// Check ParCmd.Offset.Config.Shoulder valid ? 
IF (( ParCmd.Offset.Config.Shoulder <> ArmConfigShoulder.USE_CONFIG ) AND  
    ( ParCmd.Offset.Config.Shoulder <> ArmConfigShoulder.SAME       ) AND
    ( ParCmd.Offset.Config.Shoulder <> ArmConfigShoulder.FREE       ) AND
    ( ParCmd.Offset.Config.Shoulder <> ArmConfigShoulder.BACK       ) AND
    ( ParCmd.Offset.Config.Shoulder <> ArmConfigShoulder.FRONT      ))
THEN
  // Parameter not valid
  CheckParameterValid := FALSE;
  // Set error
  SetError( ErrorID := RobotLibraryErrorIdEnum.ERR_CONFIGMODE_SHOULDER_INVALID, Overwrite := TRUE );
  // Create log entry
  CreateLogMessagePara1 ( Timestamp   := AxesGroup.State.SystemTime,
                          MessageType := MessageType.CMD,
                          Severity    := Severity.ERROR,
                          MessageCode := ErrorID,
                          MessageText := 'Invalid Parameter ParCmd.Offset.Config.Shoulder = {1}',
                          Para1       :=  ARM_CONFIG_SHOULDER_TO_STRING(ParCmd.Offset.Config.Shoulder));
  RETURN;                          
END_IF


// Check ParCmd.Offset.Config.Elbow valid ? 
IF (( ParCmd.Offset.Config.Elbow <> ArmConfigElbow.USE_CONFIG ) AND  
    ( ParCmd.Offset.Config.Elbow <> ArmConfigElbow.SAME       ) AND
    ( ParCmd.Offset.Config.Elbow <> ArmConfigElbow.FREE       ) AND
    ( ParCmd.Offset.Config.Elbow <> ArmConfigElbow.DOWN       ) AND
    ( ParCmd.Offset.Config.Elbow <> ArmConfigElbow.UP         ))
THEN
  // Parameter not valid
  CheckParameterValid := FALSE;
  // Set error
  SetError( ErrorID := RobotLibraryErrorIdEnum.ERR_CONFIGMODE_ELBOW_INVALID, Overwrite := TRUE );
  // Create log entry
  CreateLogMessagePara1 ( Timestamp   := AxesGroup.State.SystemTime,
                          MessageType := MessageType.CMD,
                          Severity    := Severity.ERROR,
                          MessageCode := ErrorID,
                          MessageText := 'Invalid Parameter ParCmd.Offset.Config.Elbow = {1}',
                          Para1       :=  ARM_CONFIG_ELBOW_TO_STRING(ParCmd.Offset.Config.Elbow));
  RETURN;                          
END_IF


// Check ParCmd.Offset.Config.Wrist valid ? 
IF (( ParCmd.Offset.Config.Wrist <> ArmConfigWrist.USE_CONFIG ) AND  
    ( ParCmd.Offset.Config.Wrist <> ArmConfigWrist.SAME       ) AND
    ( ParCmd.Offset.Config.Wrist <> ArmConfigWrist.FREE       ) AND
    ( ParCmd.Offset.Config.Wrist <> ArmConfigWrist.FLIP       ) AND
    ( ParCmd.Offset.Config.Wrist <> ArmConfigWrist.NON_FLIP   ))
THEN
  // Parameter not valid
  CheckParameterValid := FALSE;
  // Set error
  SetError( ErrorID := RobotLibraryErrorIdEnum.ERR_CONFIGMODE_WRIST_INVALID, Overwrite := TRUE );
  // Create log entry
  CreateLogMessagePara1 ( Timestamp   := AxesGroup.State.SystemTime,
                          MessageType := MessageType.CMD,
                          Severity    := Severity.ERROR,
                          MessageCode := ErrorID,
                          MessageText := 'Invalid Parameter ParCmd.Offset.Config.Wrist = {1}',
                          Para1       :=  ARM_CONFIG_WRIST_TO_STRING(ParCmd.Offset.Config.Wrist));
  RETURN;                          
END_IF


// Check ParCmd.ReferenceType valid ? 
IF (( ParCmd.ReferenceType <> ReferenceType.TOOL  ) AND
    ( ParCmd.ReferenceType <> ReferenceType.FRAME ))  
THEN
  // Parameter not valid
  CheckParameterValid := FALSE;
  // Set error
  SetError( ErrorID := RobotLibraryErrorIdEnum.ERR_INVALID_PAR_CMD, Overwrite := TRUE );
  // Create log entry
  CreateLogMessagePara1 ( Timestamp   := AxesGroup.State.SystemTime,
                          MessageType := MessageType.CMD,
                          Severity    := Severity.ERROR,
                          MessageCode := ErrorID,
                          MessageText := 'Invalid Parameter ParCmd.ReferenceType = {1}',
                          Para1       := REFERENCE_TYPE_TO_STRING(ParCmd.ReferenceType));
  RETURN;                          
END_IF


// Check ParCmd.VelocityDiffRate valid ? 
IF  (( SysDepIsValidReal(ParCmd.VelocityDiffRate) = FALSE )  OR
    ((                   ParCmd.VelocityDiffRate  <     0 )  AND 
     (                   ParCmd.VelocityDiffRate <>    -1 )) OR   
     (                   ParCmd.VelocityDiffRate  >   100 ))      
THEN
  // Parameter not valid
  CheckParameterValid := FALSE;
  // Set error
  SetError( ErrorID := RobotLibraryErrorIdEnum.ERR_INVALID_PAR_CMD, Overwrite := TRUE );
  // Create log entry
  CreateLogMessagePara1 ( Timestamp   := AxesGroup.State.SystemTime,
                          MessageType := MessageType.CMD,
                          Severity    := Severity.ERROR,
                          MessageCode := ErrorID,
                          MessageText := 'Invalid Parameter ParCmd.VelocityDiffRate = {1}',
                          Para1       := VALID_REAL_TO_STRING(ParCmd.VelocityDiffRate));                            
  RETURN;
END_IF


// Check ParCmd.AccelerationDiffRate valid ? 
IF  (( SysDepIsValidReal(ParCmd.AccelerationDiffRate) = FALSE )  OR
    ((                   ParCmd.AccelerationDiffRate  <     0 )  AND 
     (                   ParCmd.AccelerationDiffRate <>    -1 )) OR   
     (                   ParCmd.AccelerationDiffRate  >   100 ))      
THEN
  // Parameter not valid
  CheckParameterValid := FALSE;
  // Set error
  SetError( ErrorID := RobotLibraryErrorIdEnum.ERR_ACCELERATION_INVALID, Overwrite := TRUE );
  // Create log entry
  CreateLogMessagePara1 ( Timestamp   := AxesGroup.State.SystemTime,
                          MessageType := MessageType.CMD,
                          Severity    := Severity.ERROR,
                          MessageCode := ErrorID,
                          MessageText := 'Invalid Parameter ParCmd.AccelerationDiffRate = {1}',
                          Para1       := VALID_REAL_TO_STRING(ParCmd.AccelerationDiffRate));                            
  RETURN;
END_IF


// Check ParCmd.DecelerationDiffRate valid ? 
IF  (( SysDepIsValidReal(ParCmd.DecelerationDiffRate) = FALSE )  OR
    ((                   ParCmd.DecelerationDiffRate  <     0 )  AND 
     (                   ParCmd.DecelerationDiffRate <>    -1 )) OR   
     (                   ParCmd.DecelerationDiffRate  >   100 ))      
THEN
  // Parameter not valid
  CheckParameterValid := FALSE;
  // Set error
  SetError( ErrorID := RobotLibraryErrorIdEnum.ERR_DECELERATION_INVALID, Overwrite := TRUE );
  // Create log entry
  CreateLogMessagePara1 ( Timestamp   := AxesGroup.State.SystemTime,
                          MessageType := MessageType.CMD,
                          Severity    := Severity.ERROR,
                          MessageCode := ErrorID,
                          MessageText := 'Invalid Parameter ParCmd.DecelerationDiffRate = {1}',
                          Para1       := VALID_REAL_TO_STRING(ParCmd.DecelerationDiffRate));                            
  RETURN;
END_IF


// Check ParCmd.JerkDiffRate valid ? 
IF  (( SysDepIsValidReal(ParCmd.JerkDiffRate) = FALSE )  OR
    ((                   ParCmd.JerkDiffRate  <     0 )  AND 
     (                   ParCmd.JerkDiffRate <>    -1 )) OR   
     (                   ParCmd.JerkDiffRate  >   100 ))      
THEN
  // Parameter not valid
  CheckParameterValid := FALSE;
  // Set error
  SetError( ErrorID := RobotLibraryErrorIdEnum.ERR_JERK_INVALID, Overwrite := TRUE );
  // Create log entry
  CreateLogMessagePara1 ( Timestamp   := AxesGroup.State.SystemTime,
                          MessageType := MessageType.CMD,
                          Severity    := Severity.ERROR,
                          MessageCode := ErrorID,
                          MessageText := 'Invalid Parameter ParCmd.JerkDiffRate = {1}',
                          Para1       := VALID_REAL_TO_STRING(ParCmd.JerkDiffRate));                            
  RETURN;
END_IF


// Check ParCmd.ToolNo valid ? 
IF (( ParCmd.ToolNo <   0                                                ) OR   
    ( ParCmd.ToolNo > 254                                                ) OR
    ( ParCmd.ToolNo > AxesGroup.State.ConfigurationData.HighestToolIndex ) OR
    ( ParCmd.ToolNo > AxesGroup.State.UnifiedToolIndex                   ))
THEN
  // Parameter not valid
  CheckParameterValid := FALSE;
  
  // Check ToolNo available on RC ? 
  IF ( ParCmd.ToolNo > AxesGroup.State.ConfigurationData.HighestToolIndex )
  THEN
    SetError( ErrorID := RobotLibraryErrorIdEnum.ERR_TOOLNO_UNAVAILABLE, Overwrite := TRUE );
  ELSE
    SetError( ErrorID := RobotLibraryErrorIdEnum.ERR_TOOLNO_RANGE, Overwrite := TRUE );
	END_IF  
  
  // Create log entry
  CreateLogMessagePara1 ( Timestamp   := AxesGroup.State.SystemTime,
                          MessageType := MessageType.CMD,
                          Severity    := Severity.ERROR,
                          MessageCode := ErrorID,
                          MessageText := 'Invalid Parameter ParCmd.ToolNo = {1}',
                          Para1       := USINT_TO_STRING(ParCmd.ToolNo));                            
  RETURN;
END_IF


// Check ParCmd.FrameNo valid ? 
IF (( ParCmd.FrameNo <   0                                                 ) OR   
    ( ParCmd.FrameNo > 254                                                 ) OR
    ( ParCmd.FrameNo > AxesGroup.State.ConfigurationData.HighestFrameIndex ) OR
    ( ParCmd.FrameNo > AxesGroup.State.UnifiedFrameIndex                   ))         
THEN
  // Parameter not valid
  CheckParameterValid := FALSE;

  // Check FrameNo available on RC ? 
  IF ( ParCmd.FrameNo > AxesGroup.State.ConfigurationData.HighestFrameIndex )
  THEN
    SetError( ErrorID := RobotLibraryErrorIdEnum.ERR_FRAMENO_UNAVAILABLE, Overwrite := TRUE );
  ELSE
    SetError( ErrorID := RobotLibraryErrorIdEnum.ERR_FRAMENO_RANGE, Overwrite := TRUE );
	END_IF  
  
  // Create log entry
  CreateLogMessagePara1 ( Timestamp   := AxesGroup.State.SystemTime,
                          MessageType := MessageType.CMD,
                          Severity    := Severity.ERROR,
                          MessageCode := ErrorID,
                          MessageText := 'Invalid Parameter ParCmd.FrameNo = {1}',
                          Para1       := USINT_TO_STRING(ParCmd.FrameNo));                            
  RETURN;
END_IF


// Check ParCmd.InterpolationMode valid ? 
IF  (( ParCmd.InterpolationMode <> InterpolationMode.Linear_interpolation ) AND
     ( ParCmd.InterpolationMode <> InterpolationMode.Direct_interpolation ))     
THEN
  // Parameter not valid
  CheckParameterValid := FALSE;
  // Set error
  SetError( ErrorID := RobotLibraryErrorIdEnum.ERR_INVALID_PAR_CMD, Overwrite := TRUE );
  // Create log entry
  CreateLogMessagePara1 ( Timestamp   := AxesGroup.State.SystemTime,
                          MessageType := MessageType.CMD,
                          Severity    := Severity.ERROR,
                          MessageCode := ErrorID,
                          MessageText := 'Invalid Parameter ParCmd.InterpolationMode = {1}',
                          Para1       := INTERPOLATION_MODE_TO_STRING(ParCmd.InterpolationMode));
  RETURN;
END_IF
                
END_METHOD

METHOD INTERNAL CreateCommandPayload : RobotLibraryCommandDataFB
VAR_IN_OUT
  /// Robot assignment of function
  AxesGroup : AxesGroup; 
END_VAR
VAR
  /// Parameter count
 _parameterCnt : DINT;
END_VAR
// Table 6-470: Sent CMD payload (PLC to RC) of "MoveSuperImposedDynamic"
// --------------------------
// Header
// --------------------------
// Byte 00 : UINT  - Type HB     
// Byte 01 :       - Type LB    
// Byte 02 : USINT - Reserve | ExecutionMode
// Byte 03 : USINT - ParSeq  | Priority
// --------------------------
// Datablock
// --------------------------
// Byte 00 : UINT  Type;
// Byte 01 :       Type;
// Byte 02 : USINT Reserved ExecutionMode;
// Byte 03 : USINT ParSeq Priority;
// Byte 04 : UINT  VelocityRate;
// Byte 05 :       VelocityRate;
// Byte 06 :       VelocityRate;
// Byte 07 : UINT  AccelerationRate;
// Byte 08 :       AccelerationRate;
// Byte 09 :       AccelerationRate;
// Byte 10 : UINT  DecelerationRate;
// Byte 11 :       DecelerationRate;
// Byte 12 :       DecelerationRate;
// Byte 13 : UINT  JerkRate;
// Byte 14 :       JerkRate;
// Byte 15 :       JerkRate;
// Byte 16 : USINT ToolNo;
// Byte 17 : USINT FrameNo;
// Byte 18 : REAL  X;
// Byte 19 :       X;
// Byte 20 :       X;
// Byte 21 :       X;
// Byte 22 : REAL  Offset.X;
// Byte 23 :       Offset.X;
// Byte 24 :       Offset.X;
// Byte 25 :       Offset.X;
// Byte 26 : REAL  Offset.Y;
// Byte 27 :       Offset.Y;
// Byte 28 :       Offset.Y;
// Byte 29 :       Offset.Y;
// Byte 30 : REAL  Offset.Z;
// Byte 31 :       Offset.Z;
// Byte 32 :       Offset.Z;
// Byte 33 :       Offset.Z;
// Byte 34 : REAL  Offset.RX;
// Byte 35 :       Offset.RX;
// Byte 36 :       Offset.RX;
// Byte 37 :       Offset.RX;
// Byte 38 : REAL  Offset.RY;
// Byte 39 :       Offset.RY;
// Byte 40 :       Offset.RY;
// Byte 41 :       Offset.RY;
// Byte 42 : BYTE  - - - - - W E S;
// Byte 43 : BYTE  Reserved;
// Byte 44 : BYTE  Offset.TurnNumber[0];
// Byte 45 : BYTE  Offset.TurnNumber[1];
// Byte 46 : BYTE  Offset.TurnNumber[2];
// Byte 47 : BYTE  Offset.TurnNumber[3];
// Byte 48 : REAL  Offset.E1;
// Byte 49 :       Offset.E1;
// Byte 50 :       Offset.E1;
// Byte 51 :       Offset.E1;
// Byte 52 : USINT ReferenceType;
// Byte 53 : USINT InterpolationMode;
// Byte 54 : REAL  Offset.E2;
// Byte 55 :       Offset.E2;
// Byte 56 :       Offset.E2;
// Byte 57 :       Offset.E2;
// Byte 58 : REAL  Offset.E3;
// Byte 59 :       Offset.E3;
// Byte 60 :       Offset.E3;
// Byte 61 :       Offset.E3;
// Byte 62 : REAL  Offset.E4;
// Byte 63 :       Offset.E4;
// Byte 64 :       Offset.E4;
// Byte 65 :       Offset.E4;
// Byte 66 : REAL  Offset.E5;
// Byte 67 :       Offset.E5;
// Byte 68 :       Offset.E5;
// Byte 69 :       Offset.E5;
// Byte 70 : REAL  Offset.E6;
// Byte 71 :       Offset.E6;
// Byte 72 :       Offset.E6;
// Byte 73 :       Offset.E6;
                  // set command parameter 
_command.CmdTyp               :=  CmdType.MoveSuperImposedDynamic;
_command.ExecMode             :=  ExecMode;
_command.ParSeq               := _command.ParSeq;
_command.Priority             :=  Priority;
_command.VelocityDiffRate     :=  REAL_TO_PERCENT_UINT(_parCmd.VelocityDiffRate     , IsOptional := FALSE);
_command.AccelerationDiffRate :=  REAL_TO_PERCENT_UINT(_parCmd.AccelerationDiffRate , IsOptional := FALSE);
_command.DecelerationDiffRate :=  REAL_TO_PERCENT_UINT(_parCmd.DecelerationDiffRate , IsOptional := TRUE );
_command.JerkDiffRate         :=  REAL_TO_PERCENT_UINT(_parCmd.JerkDiffRate         , IsOptional := TRUE );
_command.ToolNo               := _parCmd.ToolNo;
_command.FrameNo              := _parCmd.FrameNo;
_command.Reserve_X            :=  0.0;
_command.Offset               := _parCmd.Offset;
_command.ReferenceType        := _parCmd.ReferenceType;
_command.InterpolationMode    := _parCmd.InterpolationMode;

// copy command data to header
_cmdHeader := _command;
// call base implementation to copy header to payload buffer
CreateCommandPayload := SUPER^.CreateCommandPayload(AxesGroup := AxesGroup);


// Check parameter must be added ? 
IF ( CheckAddParameter(CreateCommandPayload.PayloadPtr))
THEN
  // add command.VelocityDiffRate
  CreateCommandPayload.AddUint(_command.VelocityDiffRate);
  // inc parameter counter
 _parameterCnt := _parameterCnt + 1;  
END_IF


IF ( CheckAddParameter(CreateCommandPayload.PayloadPtr))
THEN
  // add command.AccelerationDiffRate
  CreateCommandPayload.AddUint(_command.AccelerationDiffRate);
  // inc parameter counter
 _parameterCnt := _parameterCnt + 1;  
END_IF


IF ( CheckAddParameter(CreateCommandPayload.PayloadPtr))
THEN
  // add command.DecelerationDiffRate
  CreateCommandPayload.AddUint(_command.DecelerationDiffRate);
  // inc parameter counter
 _parameterCnt := _parameterCnt + 1;  
END_IF


IF ( CheckAddParameter(CreateCommandPayload.PayloadPtr))
THEN
  // add command.JerkDiffRate
  CreateCommandPayload.AddUint(_command.JerkDiffRate);
  // inc parameter counter
 _parameterCnt := _parameterCnt + 1;  
END_IF


IF ( CheckAddParameter(CreateCommandPayload.PayloadPtr))
THEN
  // add command.ToolNo
  CreateCommandPayload.AddUsint(_command.ToolNo);
  // inc parameter counter
 _parameterCnt := _parameterCnt + 1;  
END_IF


IF ( CheckAddParameter(CreateCommandPayload.PayloadPtr))
THEN
  // add command.FrameNo
  CreateCommandPayload.AddUsint(_command.FrameNo);
  // inc parameter counter
 _parameterCnt := _parameterCnt + 1;  
END_IF


IF ( CheckAddParameter(CreateCommandPayload.PayloadPtr))
THEN
  // add command.Reserve_X
  CreateCommandPayload.AddReal(_command.Reserve_X);
  // inc parameter counter
 _parameterCnt := _parameterCnt + 1;  
END_IF


IF ( CheckAddParameter(CreateCommandPayload.PayloadPtr))
THEN
  // add command.Offset.X
  CreateCommandPayload.AddReal(_command.Offset.X);
  // inc parameter counter
 _parameterCnt := _parameterCnt + 1;  
END_IF


IF ( CheckAddParameter(CreateCommandPayload.PayloadPtr))
THEN
  // add command.Offset.Y
  CreateCommandPayload.AddReal(_command.Offset.Y);
  // inc parameter counter
 _parameterCnt := _parameterCnt + 1;  
END_IF


IF ( CheckAddParameter(CreateCommandPayload.PayloadPtr))
THEN
  // add command.Offset.Z
  CreateCommandPayload.AddReal(_command.Offset.Z);
  // inc parameter counter
 _parameterCnt := _parameterCnt + 1;  
END_IF


IF ( CheckAddParameter(CreateCommandPayload.PayloadPtr))
THEN
  // add command.Offset.Rx
  CreateCommandPayload.AddReal(_command.Offset.Rx);
  // inc parameter counter
 _parameterCnt := _parameterCnt + 1;  
END_IF


IF ( CheckAddParameter(CreateCommandPayload.PayloadPtr))
THEN
  // add command.Offset.Ry
  CreateCommandPayload.AddReal(_command.Offset.Ry);
  // inc parameter counter
 _parameterCnt := _parameterCnt + 1;  
END_IF


IF ( CheckAddParameter(CreateCommandPayload.PayloadPtr))
THEN
  // add command.Offset.Rz
  CreateCommandPayload.AddReal(_command.Offset.Rz);
  // inc parameter counter
 _parameterCnt := _parameterCnt + 1;  
END_IF


IF ( CheckAddParameter(CreateCommandPayload.PayloadPtr))
THEN
  // add command.Offset.Config
  CreateCommandPayload.AddArmConfig(_command.Offset.Config);
  // inc parameter counter
 _parameterCnt := _parameterCnt + 1;  
END_IF


IF ( CheckAddParameter(CreateCommandPayload.PayloadPtr))
THEN
  // add command.Offset.TurnNumber
  CreateCommandPayload.AddTurnNumber(_command.Offset.TurnNumber);
  // inc parameter counter
 _parameterCnt := _parameterCnt + 1;  
END_IF


IF ( CheckAddParameter(CreateCommandPayload.PayloadPtr))
THEN
  // add command.Offset.E1
  CreateCommandPayload.AddReal(_command.Offset.E1);
  // inc parameter counter
 _parameterCnt := _parameterCnt + 1;  
END_IF


IF ( CheckAddParameter(CreateCommandPayload.PayloadPtr))
THEN
  // add command.ReferenceType
  CreateCommandPayload.AddUsint(_command.ReferenceType);
  // inc parameter counter
 _parameterCnt := _parameterCnt + 1;  
END_IF


IF ( CheckAddParameter(CreateCommandPayload.PayloadPtr))
THEN
  // add command.InterpolationMode
  CreateCommandPayload.AddUsint(_command.InterpolationMode);
  // inc parameter counter
 _parameterCnt := _parameterCnt + 1;  
END_IF


IF ( CheckAddParameter(CreateCommandPayload.PayloadPtr))
THEN
  // add command.Offset.E2
  CreateCommandPayload.AddReal(_command.Offset.E2);
  // inc parameter counter
 _parameterCnt := _parameterCnt + 1;  
END_IF


IF ( CheckAddParameter(CreateCommandPayload.PayloadPtr))
THEN
  // add command.Offset.E3
  CreateCommandPayload.AddReal(_command.Offset.E3);
  // inc parameter counter
 _parameterCnt := _parameterCnt + 1;  
END_IF


IF ( CheckAddParameter(CreateCommandPayload.PayloadPtr))
THEN
  // add command.Offset.E4
  CreateCommandPayload.AddReal(_command.Offset.E4);
  // inc parameter counter
 _parameterCnt := _parameterCnt + 1;  
END_IF


IF ( CheckAddParameter(CreateCommandPayload.PayloadPtr))
THEN
  // add command.Offset.E5
  CreateCommandPayload.AddReal(_command.Offset.E5);
  // inc parameter counter
 _parameterCnt := _parameterCnt + 1;  
END_IF


IF ( CheckAddParameter(CreateCommandPayload.PayloadPtr))
THEN
  // add command.Offset.E6
  CreateCommandPayload.AddReal(_command.Offset.E6);
  // inc parameter counter
 _parameterCnt := _parameterCnt + 1;  
END_IF

  
// Create logging
CreateCommandPayloadLog(AxesGroup := AxesGroup, ParameterCnt := _parameterCnt);
                
END_METHOD

METHOD INTERNAL CreateCommandPayloadLog
VAR_IN_OUT
  /// Robot assignment of function
  AxesGroup : AxesGroup; 
END_VAR
VAR_INPUT
  /// Parameter count
  ParameterCnt : DINT;
END_VAR
VAR 
  /// internal index for loops
 _idx : DINT;
END_VAR
                  // Create log entry for Parameter start
CreateLogMessagePara1 ( Timestamp   := AxesGroup.State.SystemTime,
                        MessageType := MessageType.CMD,
                        Severity    := Severity.DEBUG,
                        MessageCode := 0,
                        MessageText := 'Create command payload with {1} parameter(s) :',
                        Para1       := DINT_TO_STRING(ParameterCnt));
  

// Return if no parameter is remaining...
IF ( ParameterCnt = 0 ) THEN RETURN; END_IF
// dec remaining parameter(s)                        
ParameterCnt := ParameterCnt - 1;
// Create log entry for VelocityDiffRate
CreateLogMessagePara1 ( Timestamp   := AxesGroup.State.SystemTime,
                        MessageType := MessageType.CMD,
                        Severity    := Severity.DEBUG,
                        MessageCode := 0,
                        MessageText := 'Command.VelocityDiffRate = {1}',
                        Para1       :=  UINT_TO_STRING(_command.VelocityDiffRate));


// Return if no parameter is remaining...
IF ( ParameterCnt = 0 ) THEN RETURN; END_IF
// dec remaining parameter(s)                        
ParameterCnt := ParameterCnt - 1;
// Create log entry for AccelerationDiffRate
CreateLogMessagePara1 ( Timestamp   := AxesGroup.State.SystemTime,
                        MessageType := MessageType.CMD,
                        Severity    := Severity.DEBUG,
                        MessageCode := 0,
                        MessageText := 'Command.AccelerationDiffRate = {1}',
                        Para1       :=  UINT_TO_STRING(_command.AccelerationDiffRate));
                        

// Return if no parameter is remaining...
IF ( ParameterCnt = 0 ) THEN RETURN; END_IF
// dec remaining parameter(s)                        
ParameterCnt := ParameterCnt - 1;
// Create log entry for DecelerationDiffRate
CreateLogMessagePara1 ( Timestamp   := AxesGroup.State.SystemTime,
                        MessageType := MessageType.CMD,
                        Severity    := Severity.DEBUG,
                        MessageCode := 0,
                        MessageText := 'Command.DecelerationDiffRate = {1}',
                        Para1       :=  UINT_TO_STRING(_command.DecelerationDiffRate));


// Return if no parameter is remaining...
IF ( ParameterCnt = 0 ) THEN RETURN; END_IF
// dec remaining parameter(s)                        
ParameterCnt := ParameterCnt - 1;
// Create log entry for JerkDiffRate
CreateLogMessagePara1 ( Timestamp   := AxesGroup.State.SystemTime,
                        MessageType := MessageType.CMD,
                        Severity    := Severity.DEBUG,
                        MessageCode := 0,
                        MessageText := 'Command.JerkDiffRate = {1}',
                        Para1       :=  UINT_TO_STRING(_command.JerkDiffRate));


// Return if no parameter is remaining...
IF ( ParameterCnt = 0 ) THEN RETURN; END_IF
// dec remaining parameter(s)                        
ParameterCnt := ParameterCnt - 1;
// Create log entry for ToolNo
CreateLogMessagePara1 ( Timestamp   := AxesGroup.State.SystemTime,
                        MessageType := MessageType.CMD,
                        Severity    := Severity.DEBUG,
                        MessageCode := 0,
                        MessageText := 'Command.ToolNo = {1}',
                        Para1       :=  USINT_TO_STRING(_command.ToolNo));


// Return if no parameter is remaining...
IF ( ParameterCnt = 0 ) THEN RETURN; END_IF
// dec remaining parameter(s)                        
ParameterCnt := ParameterCnt - 1;
// Create log entry for FrameNo
CreateLogMessagePara1 ( Timestamp   := AxesGroup.State.SystemTime,
                        MessageType := MessageType.CMD,
                        Severity    := Severity.DEBUG,
                        MessageCode := 0,
                        MessageText := 'Command.FrameNo = {1}',
                        Para1       :=  USINT_TO_STRING(_command.FrameNo));


// Return if no parameter is remaining...
IF ( ParameterCnt = 0 ) THEN RETURN; END_IF
// dec remaining parameter(s)                        
ParameterCnt := ParameterCnt - 1;
// Create log entry for Reserve_X
CreateLogMessagePara1 ( Timestamp   := AxesGroup.State.SystemTime,
                        MessageType := MessageType.CMD,
                        Severity    := Severity.DEBUG,
                        MessageCode := 0,
                        MessageText := 'Command.Reserve_X = {1}',
                        Para1       :=  REAL_TO_STRING(_command.Reserve_X));


// Return if no parameter is remaining...
IF ( ParameterCnt = 0 ) THEN RETURN; END_IF
// dec remaining parameter(s)                        
ParameterCnt := ParameterCnt - 1;
// Create log entry for Offset.X
CreateLogMessagePara1 ( Timestamp   := AxesGroup.State.SystemTime,
                        MessageType := MessageType.CMD,
                        Severity    := Severity.DEBUG,
                        MessageCode := 0,
                        MessageText := 'Command.Offset.X = {1}',
                        Para1       :=  REAL_TO_STRING(_command.Offset.X));


// Return if no parameter is remaining...
IF ( ParameterCnt = 0 ) THEN RETURN; END_IF
// dec remaining parameter(s)                        
ParameterCnt := ParameterCnt - 1;
// Create log entry for Offset.Y
CreateLogMessagePara1 ( Timestamp   := AxesGroup.State.SystemTime,
                        MessageType := MessageType.CMD,
                        Severity    := Severity.DEBUG,
                        MessageCode := 0,
                        MessageText := 'Command.Offset.Y = {1}',
                        Para1       :=  REAL_TO_STRING(_command.Offset.Y));


// Return if no parameter is remaining...
IF ( ParameterCnt = 0 ) THEN RETURN; END_IF
// dec remaining parameter(s)                        
ParameterCnt := ParameterCnt - 1;
// Create log entry for Offset.Z
CreateLogMessagePara1 ( Timestamp   := AxesGroup.State.SystemTime,
                        MessageType := MessageType.CMD,
                        Severity    := Severity.DEBUG,
                        MessageCode := 0,
                        MessageText := 'Command.Offset.Z = {1}',
                        Para1       :=  REAL_TO_STRING(_command.Offset.Z));


// Return if no parameter is remaining...
IF ( ParameterCnt = 0 ) THEN RETURN; END_IF
// dec remaining parameter(s)                        
ParameterCnt := ParameterCnt - 1;
// Create log entry for Offset.Rx
CreateLogMessagePara1 ( Timestamp   := AxesGroup.State.SystemTime,
                        MessageType := MessageType.CMD,
                        Severity    := Severity.DEBUG,
                        MessageCode := 0,
                        MessageText := 'Command.Offset.Rx = {1}',
                        Para1       :=  REAL_TO_STRING(_command.Offset.Rx));


// Return if no parameter is remaining...
IF ( ParameterCnt = 0 ) THEN RETURN; END_IF
// dec remaining parameter(s)                        
ParameterCnt := ParameterCnt - 1;
// Create log entry for Offset.Ry
CreateLogMessagePara1 ( Timestamp   := AxesGroup.State.SystemTime,
                        MessageType := MessageType.CMD,
                        Severity    := Severity.DEBUG,
                        MessageCode := 0,
                        MessageText := 'Command.Offset.Ry = {1}',
                        Para1       :=  REAL_TO_STRING(_command.Offset.Ry));


// Return if no parameter is remaining...
IF ( ParameterCnt = 0 ) THEN RETURN; END_IF
// dec remaining parameter(s)                        
ParameterCnt := ParameterCnt - 1;
// Create log entry for Offset.Rz
CreateLogMessagePara1 ( Timestamp   := AxesGroup.State.SystemTime,
                        MessageType := MessageType.CMD,
                        Severity    := Severity.DEBUG,
                        MessageCode := 0,
                        MessageText := 'Command.Offset.Rz = {1}',
                        Para1       :=  REAL_TO_STRING(_command.Offset.Rz));


// Return if no parameter is remaining...
IF ( ParameterCnt = 0 ) THEN RETURN; END_IF
// dec remaining parameter(s)                        
ParameterCnt := ParameterCnt - 1;
// Create log entry for Offset.Config
CreateLogMessagePara1 ( Timestamp   := AxesGroup.State.SystemTime,
                        MessageType := MessageType.CMD,
                        Severity    := Severity.DEBUG,
                        MessageCode := 0,
                        MessageText := 'Command.Offset.Config = {1}',
                        Para1       :=  ARM_CONFIG_TO_STRING(_command.Offset.Config));


// Return if no parameter is remaining...
IF ( ParameterCnt = 0 ) THEN RETURN; END_IF
// dec remaining parameter(s)                        
ParameterCnt := ParameterCnt - 1;
// Create log entry for Offset.TurnNumber[0]
CreateLogMessagePara1 ( Timestamp   := AxesGroup.State.SystemTime,
                        MessageType := MessageType.CMD,
                        Severity    := Severity.DEBUG,
                        MessageCode := 0,
                        MessageText := 'Command.Offset.TurnNumber[0] = {1}',
                        Para1       :=  BYTE_TO_STRING(CombineHalfSints(HalfSintHi := _command.Offset.TurnNumber.J2Turns,
                                                                        HalfSintLo := _command.Offset.TurnNumber.J1Turns)));


// Return if no parameter is remaining...
IF ( ParameterCnt = 0 ) THEN RETURN; END_IF
// dec remaining parameter(s)                        
ParameterCnt := ParameterCnt - 1;
// Create log entry for Offset.TurnNumber[1]
CreateLogMessagePara1 ( Timestamp   := AxesGroup.State.SystemTime,
                        MessageType := MessageType.CMD,
                        Severity    := Severity.DEBUG,
                        MessageCode := 0,
                        MessageText := 'Command.Offset.TurnNumber[1] = {1}',
                        Para1       :=  BYTE_TO_STRING(CombineHalfSints(HalfSintHi := _command.Offset.TurnNumber.J4Turns, 
                                                                        HalfSintLo := _command.Offset.TurnNumber.J3Turns)));


// Return if no parameter is remaining...
IF ( ParameterCnt = 0 ) THEN RETURN; END_IF
// dec remaining parameter(s)                        
ParameterCnt := ParameterCnt - 1;
// Create log entry for Offset.TurnNumber[2]
CreateLogMessagePara1 ( Timestamp   := AxesGroup.State.SystemTime,
                        MessageType := MessageType.CMD,
                        Severity    := Severity.DEBUG,
                        MessageCode := 0,
                        MessageText := 'Command.Offset.TurnNumber[2] = {1}',
                        Para1       :=  BYTE_TO_STRING(CombineHalfSints(HalfSintHi := _command.Offset.TurnNumber.J6Turns, 
                                                                        HalfSintLo := _command.Offset.TurnNumber.J5Turns)));


// Return if no parameter is remaining...
IF ( ParameterCnt = 0 ) THEN RETURN; END_IF
// dec remaining parameter(s)                        
ParameterCnt := ParameterCnt - 1;
// Create log entry for Offset.TurnNumber[3]
CreateLogMessagePara1 ( Timestamp   := AxesGroup.State.SystemTime,
                        MessageType := MessageType.CMD,
                        Severity    := Severity.DEBUG,
                        MessageCode := 0,
                        MessageText := 'Command.Position.TurnNumber[3] = {1}',
                        Para1       :=  SINT_TO_STRING(_command.Offset.TurnNumber.E1Turns));


// Return if no parameter is remaining...
IF ( ParameterCnt = 0 ) THEN RETURN; END_IF
// dec remaining parameter(s)                        
ParameterCnt := ParameterCnt - 1;
// Create log entry for Offset.E1
CreateLogMessagePara1 ( Timestamp   := AxesGroup.State.SystemTime,
                        MessageType := MessageType.CMD,
                        Severity    := Severity.DEBUG,
                        MessageCode := 0,
                        MessageText := 'Command.Offset.E1 = {1}',
                        Para1       :=  REAL_TO_STRING(_command.Offset.E1));


// Return if no parameter is remaining...
IF ( ParameterCnt = 0 ) THEN RETURN; END_IF
// dec remaining parameter(s)                        
ParameterCnt := ParameterCnt - 1;
// Create log entry for ReferenceType
CreateLogMessagePara1 ( Timestamp   := AxesGroup.State.SystemTime,
                        MessageType := MessageType.CMD,
                        Severity    := Severity.DEBUG,
                        MessageCode := 0,
                        MessageText := 'Command.ReferenceType = {1}',
                        Para1       :=  REFERENCE_TYPE_TO_STRING(_command.ReferenceType));


// Return if no parameter is remaining...
IF ( ParameterCnt = 0 ) THEN RETURN; END_IF
// dec remaining parameter(s)                        
ParameterCnt := ParameterCnt - 1;
// Create log entry for InterpolationMode
CreateLogMessagePara1 ( Timestamp   := AxesGroup.State.SystemTime,
                        MessageType := MessageType.CMD,
                        Severity    := Severity.DEBUG,
                        MessageCode := 0,
                        MessageText := 'Command.InterpolationMode = {1}',
                        Para1       :=  INTERPOLATION_MODE_TO_STRING(_command.InterpolationMode));


// Return if no parameter is remaining...
IF ( ParameterCnt = 0 ) THEN RETURN; END_IF
// dec remaining parameter(s)                        
ParameterCnt := ParameterCnt - 1;
// Create log entry for Offset.E2
CreateLogMessagePara1 ( Timestamp   := AxesGroup.State.SystemTime,
                        MessageType := MessageType.CMD,
                        Severity    := Severity.DEBUG,
                        MessageCode := 0,
                        MessageText := 'Command.Offset.E2 = {1}',
                        Para1       :=  REAL_TO_STRING(_command.Offset.E2));


// Return if no parameter is remaining...
IF ( ParameterCnt = 0 ) THEN RETURN; END_IF
// dec remaining parameter(s)                        
ParameterCnt := ParameterCnt - 1;
// Create log entry for Offset.E3
CreateLogMessagePara1 ( Timestamp   := AxesGroup.State.SystemTime,
                        MessageType := MessageType.CMD,
                        Severity    := Severity.DEBUG,
                        MessageCode := 0,
                        MessageText := 'Command.Offset.E3 = {1}',
                        Para1       :=  REAL_TO_STRING(_command.Offset.E3));


// Return if no parameter is remaining...
IF ( ParameterCnt = 0 ) THEN RETURN; END_IF
// dec remaining parameter(s)                        
ParameterCnt := ParameterCnt - 1;
// Create log entry for Offset.E4
CreateLogMessagePara1 ( Timestamp   := AxesGroup.State.SystemTime,
                        MessageType := MessageType.CMD,
                        Severity    := Severity.DEBUG,
                        MessageCode := 0,
                        MessageText := 'Command.Offset.E4 = {1}',
                        Para1       :=  REAL_TO_STRING(_command.Offset.E4));


// Return if no parameter is remaining...
IF ( ParameterCnt = 0 ) THEN RETURN; END_IF
// dec remaining parameter(s)                        
ParameterCnt := ParameterCnt - 1;
// Create log entry for Offset.E5
CreateLogMessagePara1 ( Timestamp   := AxesGroup.State.SystemTime,
                        MessageType := MessageType.CMD,
                        Severity    := Severity.DEBUG,
                        MessageCode := 0,
                        MessageText := 'Command.Offset.E5 = {1}',
                        Para1       :=  REAL_TO_STRING(_command.Offset.E5));


// Return if no parameter is remaining...
IF ( ParameterCnt = 0 ) THEN RETURN; END_IF
// dec remaining parameter(s)                        
ParameterCnt := ParameterCnt - 1;
// Create log entry for Offset.E6
CreateLogMessagePara1 ( Timestamp   := AxesGroup.State.SystemTime,
                        MessageType := MessageType.CMD,
                        Severity    := Severity.DEBUG,
                        MessageCode := 0,
                        MessageText := 'Command.Offset.E6 = {1}',
                        Para1       :=  REAL_TO_STRING(_command.Offset.E6));
                
END_METHOD

METHOD FB_init : BOOL
VAR_INPUT
  /// if TRUE, the retain variables are initialized (warm start / cold start)
  bInitRetains : BOOL; 
  /// if TRUE, the instance afterwards gets moved into the copy code (online change)
  bInCopyCode  : BOOL;  
END_VAR
                  MyType := 'MC_MoveSuperImposedDynamicFB';

ExecMode := ExecutionMode.SEQUENCE_PRIMARY;
Priority := PriorityLevel.NORMAL;
                
END_METHOD

METHOD PROTECTED OnApplyOutCmd
VAR_INPUT
  /// Command message state
  State : CmdMessageState;
END_VAR
                  IF ( State = CmdMessageState.EMPTY ) 
THEN
  // Reset command outputs
  SysDepMemSet(pDest := ADR(OutCmd), Value := 0, DataLen := SIZEOF(OutCmd));         
END_IF

IF (( State = CmdMessageState.ACTIVE ) OR
    ( State = CmdMessageState.DONE   ))
THEN
  // Update results
  OutCmd.OffsetReached     := _response.OffsetReached;
  OutCmd.Progress          :=  PERCENT_UINT_TO_REAL( Value := _response.Progress, IsOptional := TRUE);
  OutCmd.RemainingDistance := _response.RemainingDistance;
END_IF
                
END_METHOD

METHOD PROTECTED OnExecRun : DINT
VAR_IN_OUT
  /// Robot assignment of function
  AxesGroup : AxesGroup; 
END_VAR
                  // call base implementation
SUPER^.OnExecRun(AxesGroup := AxesGroup);

// building rising and falling edges
_enable_R( CLK := Enable);
_enable_F( CLK := Enable);

CASE _stepCmd OF
  
  00:  IF ( _enable_R.Q ) AND ( NOT Error) 
       THEN
         // reset the rising edge
        _enable_R();       
         // reset the falling edge
        _enable_F();       
        
         // Check function is supported and parameter are valid ?
         IF (( CheckFunctionSupported( AxesGroup := AxesGroup )) AND
             ( CheckParameterValid   ( AxesGroup := AxesGroup )))
         THEN      
           // set busy flag
           Busy := TRUE;
           // Reset command outputs
           SysDepMemSet(pDest := ADR(OutCmd), Value := 0, DataLen := SIZEOF(OutCmd));         
           // apply command parameter
          _parCmd := ParCmd;
           // init parameter sequence
          _command.ParSeq := 1;
           // create command data
           CommandData := CreateCommandPayload(AxesGroup := AxesGroup);
           // Add command to active command register
          _uniqueID := AxesGroup.Acyclic.ActiveCommandRegister.AddCmd( pCommandFB := ADR(THIS^ ));     
           // set timeout
           SetTimeout(PT := _timeoutCmd, rTimer := _timerCmd);
           // inc step counter
          _stepCmd := _stepCmd + 1;
         END_IF 
       END_IF
     

  01:  // Wait for responce received
       IF ( _responseReceived )
       THEN
         // reset response received flag
        _responseReceived := FALSE;
         // update state flags
         OnUpdateStateFlags(_response.State);
         // update state flags
         OnApplyOutCmd(_response.State);
                
         // Done, Aborted or Error ?
         IF (_response.State >= CmdMessageState.DONE )
         THEN
           // set timeout
           SetTimeout(PT := _timeoutCmd, rTimer := _timerCmd);
           // inc step counter
          _stepCmd := _stepCmd + 1; 
         END_IF
       END_IF


  02: IF (NOT Enable)
      THEN
        Reset();
	    END_IF

ELSE
  // invalid step
  SetError( ErrorID := RobotLibraryErrorIdEnum.ERR_INVALID_STEP, Overwrite := TRUE );
END_CASE


// Reset FB
IF (( _enable_R.Q ) OR
    ( _enable_F.Q ))
THEN
  Reset();
END_IF
                
END_METHOD

METHOD PROTECTED OnUpdateStateFlags
VAR_INPUT
  /// Command message state
  State : CmdMessageState;
END_VAR
                  // Reset State flags
Active := FALSE;

CASE State OF

  // No operation or process is active
  CmdMessageState.EMPTY               :;
  // Created but not yet started
  CmdMessageState.CREATED             :;
  // Buffered and awaiting execution
  CmdMessageState.BUFFERED            : CommandBuffered    := TRUE;
                                        ParameterAccepted  := TRUE;
  // Buffered in planner for future execution
  CmdMessageState.BUFFERED_IN_PLANNER : CommandBuffered    := TRUE;
                                        ParameterAccepted  := TRUE;
  // Currently active and in progress
  CmdMessageState.ACTIVE              : Active             := TRUE;
                                        Enabled            := TRUE;                                  
  // Interrupted and awaiting continuation
  CmdMessageState.INTERRUPTED         :;     
  // Requested for abort
  CmdMessageState.ABORT_REQUEST       :;
  // Successfully completed
  CmdMessageState.DONE                : Busy               := FALSE;
  // Aborted before completion
  CmdMessageState.ABORTED             : Busy               := FALSE;
  // Encountered an error during execution
  CmdMessageState.ERROR               : Error              := TRUE;
                                        Busy               := FALSE;
END_CASE
                
END_METHOD

METHOD INTERNAL ParseResponsePayload : DINT
VAR_INPUT
  /// Response data
  ResponseData : RobotLibraryResponseDataFB;
  /// Timestamp
  Timestamp    : SystemTime;  
END_VAR
VAR
  /// Parameter count
 _parameterCnt : DINT;
END_VAR
// Table 6-471: Received CMD payload (RC to PLC) of "MoveSuperImposedDynamic"
// --------------------------
// Header
// --------------------------
// Byte 00 : USINT - ParSeq | State     
// Byte 01 : SINT  - AlarmMessageSeverity    
// Byte 02 : UINT  - AlarmMessageCode HB
// Byte 03 :       - AlarmMessageCode LB
// --------------------------
// Datablock
// --------------------------
// Byte 04 : UINT  - Progress HB
// Byte 05 : UINT  - Progress LB
// Byte 06 : REAL  - RemainingDistance HW HB
// Byte 07 :       - RemainingDistance HW LB
// Byte 08 :       - RemainingDistance LW HB
// Byte 09 :       - RemainingDistance LW LB
// Byte 10 : BOOL  - OffsetReached
// --------------------------
                  // call base implementation to parse the header from payload buffer
ResponseData.PayloadPtr := SUPER^.ParseResponsePayload(ResponseData := ResponseData, Timestamp := Timestamp);

// copy parsed header to response
_response.ParSeq               := _rspHeader.ParSeq;
_response.State                := _rspHeader.State;
_response.AlarmMessageSeverity := _rspHeader.AlarmMessageSeverity;
_response.AlarmMessageCode     := _rspHeader.AlarmMessageCode;


// Check payload remaining ? 
IF ( ResponseData.IsPayloadRemaining)
THEN  
  // Get Response.Progress
 _response.Progress := ResponseData.GetUint();
  // inc parameter counter
 _parameterCnt := _parameterCnt + 1;
END_IF


// Check payload remaining ? 
IF ( ResponseData.IsPayloadRemaining)
THEN  
  // Get Response.RemainingDistance
 _response.RemainingDistance := ResponseData.GetReal();
  // inc parameter counter
 _parameterCnt := _parameterCnt + 1;
END_IF
 
 
// Check payload remaining ? 
IF ( ResponseData.IsPayloadRemaining)
THEN  
  // Get Response.OffsetReached
 _response.OffsetReached := ResponseData.GetBool();
  // inc parameter counter
 _parameterCnt := _parameterCnt + 1;
END_IF

 
// Create logging
ParseResponsePayloadLog(ResponseData := ResponseData, Timestamp := Timestamp, ParameterCnt := _parameterCnt);
                
END_METHOD

METHOD INTERNAL ParseResponsePayloadLog
VAR_INPUT
  /// Response data
  ResponseData : RobotLibraryResponseDataFB;
  /// Timestamp
  Timestamp    : SystemTime;  
  /// Parameter count
  ParameterCnt : DINT;
END_VAR
                  // Create log entry for Parameter start
CreateLogMessagePara1 ( Timestamp   := Timestamp,
                        MessageType := MessageType.CMD,
                        Severity    := Severity.DEBUG,
                        MessageCode := 0,
                        MessageText := '{1} parameter(s) to parse from the response data:',
                        Para1       := DINT_TO_STRING(ParameterCnt));
                        

// Return if no parameter is remaining...
IF ( ParameterCnt = 0 ) THEN RETURN; END_IF
// dec remaining parameter(s)                        
ParameterCnt := ParameterCnt - 1;
// Create log entry for Progress
CreateLogMessagePara1 ( Timestamp   := Timestamp,
                        MessageType := MessageType.CMD,
                        Severity    := Severity.DEBUG,
                        MessageCode := 0,
                        MessageText := 'Response.Progress = {1}',
                        Para1       :=  UINT_TO_STRING(_response.Progress));


// Return if no parameter is remaining...
IF ( ParameterCnt = 0 ) THEN RETURN; END_IF
// dec remaining parameter(s)                        
ParameterCnt := ParameterCnt - 1;
// Create log entry for RemainingDistance
CreateLogMessagePara1 ( Timestamp   := Timestamp,
                        MessageType := MessageType.CMD,
                        Severity    := Severity.DEBUG,
                        MessageCode := 0,
                        MessageText := 'Response.RemainingDistance = {1}',
                        Para1       :=  REAL_TO_STRING(_response.RemainingDistance));


// Return if no parameter is remaining...
IF ( ParameterCnt = 0 ) THEN RETURN; END_IF
// dec remaining parameter(s)                        
ParameterCnt := ParameterCnt - 1;
// Create log entry for OffsetReached
CreateLogMessagePara1 ( Timestamp   := Timestamp,
                        MessageType := MessageType.CMD,
                        Severity    := Severity.DEBUG,
                        MessageCode := 0,
                        MessageText := 'Response.OffsetReached = {1}',
                        Para1       :=  BOOL_TO_STRING(_response.OffsetReached));

                
END_METHOD

METHOD PROTECTED Reset : DINT
VAR_INPUT
END_VAR
                  Reset := SUPER^.Reset();

Busy              := FALSE;
CommandBuffered   := FALSE;
Active            := FALSE;
ParameterAccepted := FALSE;
                
END_METHOD
END_FUNCTION_BLOCK

/// "Action" that initiates specified events when triggered
FUNCTION_BLOCK MC_ReactAtTriggerFB EXTENDS RobotLibraryBaseExecuteFB
// ------------------------------------------------------------------------- 
//  SRCI Robot Library                                                
// ------------------------------------------------------------------------- 
//                                                                           
//  Object:      ReactAtTriggerFB                                       
//  Author:      Thorsten Brach                                                
//  Date:        2024-06-01
//
//  Description:                                              
//   
//                                                                           
//  Copyright: 
//    (C) 2024 Thorsten Brach. All rights reserved                                                                                                                                            
//             Licensed under the MIT License.
//                                                                           
//  Disclaimer:                                                                           
//    This project is provided without any guarantee and can be used for   
//    private and commercial purposes. Any use is at the user’s 
//    own risk and responsibility.
//
// -------------------------------------------------------------------------
VAR_INPUT
  /// command parameter 
  ParCmd          : ReactAtTriggerParCmd;
  /// Processing mode
  ProcessingMode  : ProcessingMode;
END_VAR
VAR_OUTPUT
  /// Command is transferred and confirmed by the RC
  CommandBuffered : BOOL;
  /// command results
  OutCmd          : ReactAtTriggerOutCmd;     
END_VAR

VAR
  /// internal copy of command parameter 
 _parCmd          : ReactAtTriggerParCmd;
  /// command data to send
 _command         : ReactAtTriggerSendData;
  /// response data received
 _response        : ReactAtTriggerRecvData;      
END_VAR

            SUPER^(AxesGroup := AxesGroup);
          

METHOD INTERNAL CheckAddParameter : BOOL
VAR_INPUT
  /// Payload pointer
  PayloadPtr : UDINT;
END_VAR
VAR
  /// Payload as byte array
  Payload    : ARRAY [1..SIZEOF(_command)] OF BYTE;
  /// Null Byte array 
  Null       : ARRAY [1..SIZEOF(_command)] OF BYTE;
  /// Data length to compare
  DataLen    : UDINT;
END_VAR
                  // Payload pointer must be decreased by one byte, because ADR(Payload) is already one byte !
PayloadPtr := LIMIT (0, PayloadPtr - 1, SIZEOF(Payload) -1);
// Convert command struct to payload array
SysDepMemCpy( pDest := ADR(Payload), pSrc := ADR(_command), DataLen := SIZEOF(_command));
// Calculate the data length to compare - at least one byte must be compared !
DataLen := LIMIT(1, SIZEOF(Payload) - PayloadPtr, SIZEOF(Payload)); 
// Compare Payload-Array with Null-Byte-Array
CheckAddParameter := SysDepMemCmp( pData1 := ADR(Payload) + PayloadPtr , pData2 := ADR(Null), DataLen := DataLen) <>  RobotLibraryConstants.OK ;
                
END_METHOD

METHOD PROTECTED CheckFunctionSupported : BOOL
VAR_IN_OUT
  /// Robot assignment of function
  AxesGroup : AxesGroup; 
END_VAR
                  CheckFunctionSupported := AxesGroup.State.RobotData.RCSupportedFunctions.ReactAtTrigger;

IF ( NOT CheckFunctionSupported )
THEN
  // call base implementation for set error and create log entry
  SUPER^.CheckFunctionSupported(AxesGroup := AxesGroup);
END_IF
                
END_METHOD

METHOD PROTECTED CheckParameterChanged : BOOL
VAR_IN_OUT
  /// Robot assignment of function
  AxesGroup    : AxesGroup; 
END_VAR
                  // Check ParCmd Size is > 0, because MemCmp does not work correctly with size = 0
IF (SIZEOF(ParCmd) = 0) OR (_stepCmd = 0)
THEN 
  RETURN;
END_IF

// compare memory 
_parameterChanged := ( SysDepMemCmp(pData1 := ADR(ParCmd), pData2 := ADR(_parCmd), DataLen := SIZEOF(ParCmd)) <> RobotLibraryConstants.OK );

// check parameter valid ?
_parameterValid   := CheckParameterValid( AxesGroup := AxesGroup );

IF ((  _parameterChanged        )  AND 
    (  _parameterValid          )) OR
    (  _parameterUpdateInternal )  
THEN  
  // Create log entry for parameter changed event
  CreateLogMessagePara1 ( Timestamp   := AxesGroup.State.SystemTime,
                          MessageType := MessageType.CMD,
                          Severity    := Severity.DEBUG,
                          MessageCode := 0,
                          MessageText := 'NotifyParameterChanged Event {1}',
                          Para1       :=  '' );

  // reset internal flag for send parameter update
 _parameterUpdateInternal := FALSE;
  // update internal copy of parameters 
 _parCmd := ParCmd;
  // inc parameter sequence
 _command.ParSeq := _command.ParSeq + 1;
  // update command data  
  CommandData := CreateCommandPayload(AxesGroup := AxesGroup); // ( Access via reference to rCommandFB in ACR )
  // notify active command register 
  AxesGroup.Acyclic.ActiveCommandRegister.NotifyParameterChanged := _uniqueID;
END_IF
                
END_METHOD

METHOD PROTECTED CheckParameterValid : BOOL
VAR_IN_OUT
  /// Robot assignment of function
  AxesGroup : AxesGroup; 
END_VAR
VAR
  /// internal index for loops
 _idx : DINT;
END_VAR
                  CheckParameterValid := TRUE;

// Check ParCmd.ProcessingMode defined ? 
IF (( ProcessingMode < ProcessingModeEnum.BUFFERED         ) AND
    ( ProcessingMode > ProcessingModeEnum.TRIGGER_MULTIPLE ))
THEN
  // Parameter not valid
  CheckParameterValid := FALSE;
  // Set error
  SetError( ErrorID := RobotLibraryErrorIdEnum.ERR_PROCESSINGMODE_NOT_DEFINED, Overwrite := TRUE );
  // Create log entry
  CreateLogMessagePara1 ( Timestamp   := AxesGroup.State.SystemTime,
                          MessageType := MessageType.CMD,
                          Severity    := Severity.ERROR,
                          MessageCode := ErrorID,
                          MessageText := 'Invalid Parameter ParCmd.ProcessingMode = {1}',
                          Para1       := PROCESSING_MODE_TO_STRING(ProcessingMode));
  RETURN;                          
END_IF

// Check ProcessingMode valid ? 
IF (( ProcessingMode <> ProcessingModeEnum.DEACTIVATE       ) AND 
    ( ProcessingMode <> ProcessingModeEnum.TRIGGER_ONCE     ) AND  
    ( ProcessingMode <> ProcessingModeEnum.TRIGGER_MULTIPLE ))  
THEN
  // Parameter not valid
  CheckParameterValid := FALSE;
  // Set error
  SetError( ErrorID := RobotLibraryErrorIdEnum.ERR_PROCESSINGMODE_NOT_ALLOWED, Overwrite := TRUE );
  // Create log entry
  CreateLogMessagePara1 ( Timestamp   := AxesGroup.State.SystemTime,
                          MessageType := MessageType.CMD,
                          Severity    := Severity.ERROR,
                          MessageCode := ErrorID,
                          MessageText := 'Invalid Parameter ProcessingMode = {1}',
                          Para1       := PROCESSING_MODE_TO_STRING(ProcessingMode));
  RETURN;                          
END_IF


// Check ParCmd.ReactionMode valid ? 
IF (( ParCmd.ReactionMode <> TriggerReactionMode.NO_REACTION                ) AND
    ( ParCmd.ReactionMode <> TriggerReactionMode.INTERRUPT                  ) AND
    ( ParCmd.ReactionMode <> TriggerReactionMode.GROUP_STOP                 ) AND
    ( ParCmd.ReactionMode <> TriggerReactionMode.DISABLE_ROBOT              ) AND
    ( ParCmd.ReactionMode <> TriggerReactionMode.STOP_ACTUAL_MOTION_COMMAND ))
THEN
  // Parameter not valid
  CheckParameterValid := FALSE;
  // Set error
  SetError( ErrorID := RobotLibraryErrorIdEnum.ERR_INVALID_PAR_CMD, Overwrite := TRUE );
  // Create log entry
  CreateLogMessagePara1 ( Timestamp   := AxesGroup.State.SystemTime,
                          MessageType := MessageType.CMD,
                          Severity    := Severity.ERROR,
                          MessageCode := ErrorID,
                          MessageText := 'Invalid Parameter ParCmd.ReactionMode = {1}',
                          Para1       := TRIGGER_REACTION_MODE_TO_STRING(ParCmd.ReactionMode));
  RETURN;                          
END_IF


// Check ParCmd.ListenerID valid ? 
IF  (( ParCmd.ListenerID <   0 ) OR
     ( ParCmd.ListenerID > 127 ))     
THEN
  // Parameter not valid
  CheckParameterValid := FALSE;
  // Set error
  SetError( ErrorID := RobotLibraryErrorIdEnum.ERR_INVALID_PAR_CMD, Overwrite := TRUE );
  // Create log entry
  CreateLogMessagePara1 ( Timestamp   := AxesGroup.State.SystemTime,
                          MessageType := MessageType.CMD,
                          Severity    := Severity.ERROR,
                          MessageCode := ErrorID,
                          MessageText := 'Invalid Parameter ParCmd.ListenerID = {1}',
                          Para1       := SINT_TO_STRING(ParCmd.ListenerID));
  RETURN;
END_IF

                
END_METHOD

METHOD INTERNAL CreateCommandPayload : RobotLibraryCommandDataFB
VAR_IN_OUT
  /// Robot assignment of function
  AxesGroup : AxesGroup; 
END_VAR
VAR
  /// internal index for loops
 _idx          : DINT;
  /// Parameter count
 _parameterCnt : DINT;
END_VAR
// Table 6-604: Sent CMD payload (PLC to RC) of "ReactAtTrigger"
// --------------------------
// Header
// --------------------------
// Byte 00 : UINT  - Type HB     
// Byte 01 :       - Type LB    
// Byte 02 : USINT - Reserve | ExecutionMode
// Byte 03 : USINT - ParSeq  | Priority
// --------------------------
// Datablock
// --------------------------
// Byte 04 : SINT       - EmitterID[0]
// Byte 05 : SINT       - EmitterID[1]
// Byte 06 : SINT       - EmitterID[2]
// Byte 07 : SINT       - EmitterID[3]
// Byte 08 : SINT       - ListenerID
// Byte 09 : BYTE       - Reserved
// Byte 10 : SINT       - ReactionMode
                  // set command parameter 
_command.CmdTyp       :=  CmdType.ReactAtTrigger;
_command.ExecMode     :=  ExecMode;
_command.ParSeq       := _command.ParSeq;
_command.Priority     :=  Priority;                      
_command.EmitterID[0] := 0;
_command.EmitterID[1] := 0;
_command.EmitterID[2] := 0;
_command.EmitterID[3] := 0;
_command.ListenerID   := _parCmd.ListenerID; 
_command.Reserve      := 0;
_command.ReactionMode := _parCmd.ReactionMode;


// copy command data to header
_cmdHeader := _command;
// call base implementation to copy header to payload buffer
CreateCommandPayload := SUPER^.CreateCommandPayload(AxesGroup := AxesGroup);


FOR _idx := 0 TO 3 
DO
  // Check parameter must be added ? 
  IF ( CheckAddParameter(CreateCommandPayload.PayloadPtr))
  THEN
    // add command.EmitterID[x]
    CreateCommandPayload.AddSint(_command.EmitterID[_idx]);
    // inc parameter counter
   _parameterCnt := _parameterCnt + 1;  
  END_IF
END_FOR


// Check parameter must be added ? 
IF ( CheckAddParameter(CreateCommandPayload.PayloadPtr))
THEN
  // add command.ListenerID
  CreateCommandPayload.AddSint(_command.ListenerID);
  // inc parameter counter
 _parameterCnt := _parameterCnt + 1;  
END_IF


// Check parameter must be added ? 
IF ( CheckAddParameter(CreateCommandPayload.PayloadPtr))
THEN
  // add command.Reserve
  CreateCommandPayload.AddSint(_command.Reserve);
  // inc parameter counter
 _parameterCnt := _parameterCnt + 1;  
END_IF


// Check parameter must be added ? 
IF ( CheckAddParameter(CreateCommandPayload.PayloadPtr))
THEN
  // add command.ReactionMode
  CreateCommandPayload.AddSint(_command.ReactionMode);
  // inc parameter counter
 _parameterCnt := _parameterCnt + 1;  
END_IF


// Create logging
CreateCommandPayloadLog(AxesGroup := AxesGroup, ParameterCnt := _parameterCnt);
                
END_METHOD

METHOD INTERNAL CreateCommandPayloadLog
VAR_IN_OUT
  /// Robot assignment of function
  AxesGroup : AxesGroup; 
END_VAR
VAR_INPUT
  /// Parameter count
  ParameterCnt : DINT;
END_VAR
VAR 
  /// internal index for loops
 _idx : DINT;
END_VAR
                  // Create log entry for Parameter start
CreateLogMessagePara1 ( Timestamp   := AxesGroup.State.SystemTime,
                        MessageType := MessageType.CMD,
                        Severity    := Severity.DEBUG,
                        MessageCode := 0,
                        MessageText := 'Create command payload with {1} parameter(s) :',
                        Para1       := DINT_TO_STRING(ParameterCnt));
  
// Create log entry for EmitterID[x]
FOR _idx := 0 TO 3
DO
  // Return if no parameter is remaining...
  IF ( ParameterCnt = 0 ) THEN RETURN; END_IF
  // dec remaining parameter(s)                        
  ParameterCnt := ParameterCnt - 1;
  // Create log entry for Command.EmitterID
  CreateLogMessagePara2 ( Timestamp   := AxesGroup.State.SystemTime,
                          MessageType := MessageType.CMD,
                          Severity    := Severity.DEBUG,
                          MessageCode := 0,
                          MessageText := 'Command.EmitterID[{2}] = {1}',
                          Para1       :=  SINT_TO_STRING(_command.EmitterID[_idx]),
                          Para2       :=  DINT_TO_STRING(_idx));
END_FOR


// Return if no parameter is remaining...
IF ( ParameterCnt = 0 ) THEN RETURN; END_IF
// dec remaining parameter(s)                        
ParameterCnt := ParameterCnt - 1;
// Create log entry for ListenerID
CreateLogMessagePara1 ( Timestamp   := AxesGroup.State.SystemTime,
                        MessageType := MessageType.CMD,
                        Severity    := Severity.DEBUG,
                        MessageCode := 0,
                        MessageText := 'Command.ListenerID = {1}',
                        Para1       :=  SINT_TO_STRING(_command.ListenerID));
                        

// Return if no parameter is remaining...
IF ( ParameterCnt = 0 ) THEN RETURN; END_IF
// dec remaining parameter(s)                        
ParameterCnt := ParameterCnt - 1;
// Create log entry for Reserve
CreateLogMessagePara1 ( Timestamp   := AxesGroup.State.SystemTime,
                        MessageType := MessageType.CMD,
                        Severity    := Severity.DEBUG,
                        MessageCode := 0,
                        MessageText := 'Command.Reserve = {1}',
                        Para1       :=  SINT_TO_STRING(_command.Reserve));


// Return if no parameter is remaining...
IF ( ParameterCnt = 0 ) THEN RETURN; END_IF
// dec remaining parameter(s)                        
ParameterCnt := ParameterCnt - 1;
// Create log entry for ReactionMode
CreateLogMessagePara1 ( Timestamp   := AxesGroup.State.SystemTime,
                        MessageType := MessageType.CMD,
                        Severity    := Severity.DEBUG,
                        MessageCode := 0,
                        MessageText := 'Command.ReactionMode = {1}',
                        Para1       :=  TRIGGER_REACTION_MODE_TO_STRING(_command.ReactionMode));

                
END_METHOD

METHOD FB_init : BOOL
VAR_INPUT
  /// if TRUE, the retain variables are initialized (warm start / cold start)
  bInitRetains : BOOL; 
  /// if TRUE, the instance afterwards gets moved into the copy code (online change)
  bInCopyCode  : BOOL;  
END_VAR
                  MyType := 'MC_ReactAtTriggerFB';

ExecMode       := ExecutionMode.PARALLEL;
Priority       := PriorityLevel.NORMAL;
ProcessingMode := ProcessingModeEnum.TRIGGER_ONCE;
                
END_METHOD

METHOD PROTECTED OnApplyOutCmd
VAR_INPUT
  /// Command message state
  State : CmdMessageState;
END_VAR
                  IF ( State = CmdMessageState.EMPTY ) 
THEN
  // Reset command outputs
  SysDepMemSet(pDest := ADR(OutCmd), Value := 0, DataLen := SIZEOF(OutCmd));         
END_IF

IF (( State = CmdMessageState.ACTIVE ) OR
    ( State = CmdMessageState.DONE   ))
THEN
  // Update results
  OutCmd.InvocationCounter := _response.InvocationCounter;
  OutCmd.OriginID          := _response.OriginID;
END_IF
                
END_METHOD

METHOD PROTECTED OnExecRun : DINT
VAR_IN_OUT
  /// Robot assignment of function
  AxesGroup : AxesGroup; 
END_VAR
                  // call base implementation
SUPER^.OnExecRun(AxesGroup := AxesGroup);

CASE _stepCmd OF
  
  00:  IF ( _execute_R.Q ) AND ( NOT Error)  
       THEN
         // Check function is supported and parameter are valid ?
         IF (( CheckFunctionSupported( AxesGroup := AxesGroup )) AND
             ( CheckParameterValid   ( AxesGroup := AxesGroup )))
         THEN      
           // set busy flag
           Busy := TRUE;
           // Reset command outputs
           SysDepMemSet(pDest := ADR(OutCmd), Value := 0, DataLen := SIZEOF(OutCmd));         
           // apply command parameter
          _parCmd := ParCmd;
           // init parameter sequence
          _command.ParSeq := 1;
           // create command data
           CommandData := CreateCommandPayload(AxesGroup := AxesGroup);
           // Add command to active command register
          _uniqueID := AxesGroup.Acyclic.ActiveCommandRegister.AddCmd( pCommandFB := ADR(THIS^ ));     
           // set timeout
           SetTimeout(PT := _timeoutCmd, rTimer := _timerCmd);
           // inc step counter
          _stepCmd := _stepCmd + 1;
         END_IF 
       END_IF
     

  01:  // Wait for responce received
       IF ( _responseReceived )
       THEN
         // reset response received flag
        _responseReceived := FALSE;
         // update state flags
         OnUpdateStateFlags(_response.State);
         // update state flags
         OnApplyOutCmd(_response.State);

         // Done, Aborted or Error ?
         IF (_response.State >= CmdMessageState.DONE )
         THEN
           // set timeout
           SetTimeout(PT := _timeoutCmd, rTimer := _timerCmd);
           // inc step counter
          _stepCmd := _stepCmd + 1; 
         END_IF
       END_IF


  02: IF ( NOT Execute)
      THEN
        Reset();  
      END_IF     

ELSE
  // invalid step
  SetError( ErrorID := RobotLibraryErrorIdEnum.ERR_INVALID_STEP, Overwrite := TRUE );
END_CASE


// Reset FB
IF ( NOT Execute )
THEN
  Reset(); 
END_IF
                
END_METHOD

METHOD PROTECTED OnUpdateStateFlags
VAR_INPUT
  /// Command message state
  State : CmdMessageState;
END_VAR
                  // Reset State flags
Done := FALSE;

CASE State OF

  // No operation or process is active
  CmdMessageState.EMPTY               :;
  // Created but not yet started
  CmdMessageState.CREATED             :;
  // Buffered and awaiting execution
  CmdMessageState.BUFFERED            : CommandBuffered    := TRUE;                                        
  // Buffered in planner for future execution
  CmdMessageState.BUFFERED_IN_PLANNER : CommandBuffered    := TRUE;
  // Currently active and in progress
  CmdMessageState.ACTIVE              :;                                  
  // Interrupted and awaiting continuation
  CmdMessageState.INTERRUPTED         :;     
  // Requested for abort
  CmdMessageState.ABORT_REQUEST       :;
  // Successfully completed
  CmdMessageState.DONE                : Done               := TRUE;
                                        Busy               := FALSE;
  // Aborted before completion
  CmdMessageState.ABORTED             : Busy               := FALSE;
  // Encountered an error during execution
  CmdMessageState.ERROR               : Error              := TRUE;
                                        Busy               := FALSE;
END_CASE
                
END_METHOD

METHOD INTERNAL ParseResponsePayload : DINT
VAR_INPUT
  /// Response data
  ResponseData : RobotLibraryResponseDataFB;
  /// Timestamp
  Timestamp    : SystemTime;  
END_VAR
VAR
  /// Parameter count
 _parameterCnt : DINT;
END_VAR
// Table 6-605: Received CMD payload (RC to PLC) of "ReactAtTrigger"
// --------------------------
// Header
// --------------------------
// Byte 00 : USINT   - ParSeq | State     
// Byte 01 : SINT    - AlarmMessageSeverity    
// Byte 02 : UINT    - AlarmMessageCode HB
// Byte 03 :         - AlarmMessageCode LB
// --------------------------
// Datablock
// --------------------------
// Byte 04 : USINT   - InvocationCounter
// Byte 05 : SINT    - Reserve
// Byte 06 : INT     - OriginID LW HB
// Byte 07 :         - OriginID LW LB
                  // call base implementation to parse the header from payload buffer
ResponseData.PayloadPtr := SUPER^.ParseResponsePayload(ResponseData := ResponseData, Timestamp := Timestamp);

// copy parsed header to response
_response.ParSeq               := _rspHeader.ParSeq;
_response.State                := _rspHeader.State;
_response.AlarmMessageSeverity := _rspHeader.AlarmMessageSeverity;
_response.AlarmMessageCode     := _rspHeader.AlarmMessageCode;


// Check payload remaining ? 
IF ( ResponseData.IsPayloadRemaining)
THEN  
  // Get Response.InvocationCounter
 _response.InvocationCounter := ResponseData.GetUsint();
  // inc parameter counter
 _parameterCnt := _parameterCnt + 1;
END_IF


// Check payload remaining ? 
IF ( ResponseData.IsPayloadRemaining)
THEN  
  // Get Response.Reserve
 _response.Reserve := ResponseData.GetSint();
  // inc parameter counter
 _parameterCnt := _parameterCnt + 1;
END_IF


// Check payload remaining ? 
IF ( ResponseData.IsPayloadRemaining)
THEN  
  // Get Response.OriginID
 _response.OriginID := ResponseData.GetInt();
  // inc parameter counter
 _parameterCnt := _parameterCnt + 1;
END_IF


// Create logging
ParseResponsePayloadLog(ResponseData := ResponseData, Timestamp := Timestamp, ParameterCnt := _parameterCnt);
                
END_METHOD

METHOD INTERNAL ParseResponsePayloadLog
VAR_INPUT
  /// Response data
  ResponseData : RobotLibraryResponseDataFB;
  /// Timestamp
  Timestamp    : SystemTime;  
  /// Parameter count
  ParameterCnt : DINT;
END_VAR
                  // Create log entry for Parameter start
CreateLogMessagePara1 ( Timestamp   := Timestamp,
                        MessageType := MessageType.CMD,
                        Severity    := Severity.DEBUG,
                        MessageCode := 0,
                        MessageText := '{1} parameter(s) to parse from the response data:',
                        Para1       := DINT_TO_STRING(ParameterCnt));
                        

// Return if no parameter is remaining...
IF ( ParameterCnt = 0 ) THEN RETURN; END_IF
// dec remaining parameter(s)                        
ParameterCnt := ParameterCnt - 1;
// Create log entry for InvocationCounter
CreateLogMessagePara1 ( Timestamp   := Timestamp,
                        MessageType := MessageType.CMD,
                        Severity    := Severity.DEBUG,
                        MessageCode := 0,
                        MessageText := 'Response.InvocationCounter = {1}',
                        Para1       :=  USINT_TO_STRING(_response.InvocationCounter));


// Return if no parameter is remaining...
IF ( ParameterCnt = 0 ) THEN RETURN; END_IF
// dec remaining parameter(s)                        
ParameterCnt := ParameterCnt - 1;
// Create log entry for Reserve
CreateLogMessagePara1 ( Timestamp   := Timestamp,
                        MessageType := MessageType.CMD,
                        Severity    := Severity.DEBUG,
                        MessageCode := 0,
                        MessageText := 'Response.Reserve = {1}',
                        Para1       :=  SINT_TO_STRING(_response.Reserve));


// Return if no parameter is remaining...
IF ( ParameterCnt = 0 ) THEN RETURN; END_IF
// dec remaining parameter(s)                        
ParameterCnt := ParameterCnt - 1;
// Create log entry for OriginID
CreateLogMessagePara1 ( Timestamp   := Timestamp,
                        MessageType := MessageType.CMD,
                        Severity    := Severity.DEBUG,
                        MessageCode := 0,
                        MessageText := 'Response.OriginID = {1}',
                        Para1       :=  INT_TO_STRING(_response.OriginID));
                
END_METHOD

METHOD PROTECTED Reset : DINT
VAR_INPUT
END_VAR
                  Reset := SUPER^.Reset();

Done               := FALSE;
Busy               := FALSE;
CommandBuffered    := FALSE;  
                
END_METHOD
END_FUNCTION_BLOCK

/// Trigger "Actions" based on incoming error event
FUNCTION_BLOCK MC_SetTriggerErrorFB EXTENDS RobotLibraryBaseExecuteFB
// ------------------------------------------------------------------------- 
//  SRCI Robot Library                                                
// ------------------------------------------------------------------------- 
//                                                                           
//  Object:      SetTriggerErrorFB                                       
//  Author:      Thorsten Brach                                                
//  Date:        2024-06-01
//
//  Description:                                              
//   
//                                                                           
//  Copyright: 
//    (C) 2024 Thorsten Brach. All rights reserved                                                                                                                                            
//             Licensed under the MIT License.
//                                                                           
//  Disclaimer:                                                                           
//    This project is provided without any guarantee and can be used for   
//    private and commercial purposes. Any use is at the user’s 
//    own risk and responsibility.
//
// -------------------------------------------------------------------------
VAR_INPUT
  /// command parameter 
  ParCmd           : SetTriggerErrorParCmd;
  /// Processing mode
  ProcessingMode   : ProcessingMode;
END_VAR
VAR_OUTPUT
  /// Command is transferred and confirmed by the RC
  CommandBuffered  : BOOL;
  /// TRUE, when the monitoring of the input parameter values is active.
  MonitoringActive : BOOL;
  /// command results
  OutCmd           : SetTriggerErrorOutCmd;     
END_VAR

VAR
  /// internal copy of command parameter 
 _parCmd           : SetTriggerErrorParCmd;
  /// command data to send
 _command          : SetTriggerErrorSendData;
  /// response data received
 _response         : SetTriggerErrorRecvData;      
END_VAR

            SUPER^(AxesGroup := AxesGroup);
          

METHOD INTERNAL CheckAddParameter : BOOL
VAR_INPUT
  /// Payload pointer
  PayloadPtr : UDINT;
END_VAR
VAR
  /// Payload as byte array
  Payload    : ARRAY [1..SIZEOF(_command)] OF BYTE;
  /// Null Byte array 
  Null       : ARRAY [1..SIZEOF(_command)] OF BYTE;
  /// Data length to compare
  DataLen    : UDINT;
END_VAR
                  // Payload pointer must be decreased by one byte, because ADR(Payload) is already one byte !
PayloadPtr := LIMIT (0, PayloadPtr - 1, SIZEOF(Payload) -1);
// Convert command struct to payload array
SysDepMemCpy( pDest := ADR(Payload), pSrc := ADR(_command), DataLen := SIZEOF(_command));
// Calculate the data length to compare - at least one byte must be compared !
DataLen := LIMIT(1, SIZEOF(Payload) - PayloadPtr, SIZEOF(Payload)); 
// Compare Payload-Array with Null-Byte-Array
CheckAddParameter := SysDepMemCmp( pData1 := ADR(Payload) + PayloadPtr , pData2 := ADR(Null), DataLen := DataLen) <>  RobotLibraryConstants.OK ;
                
END_METHOD

METHOD PROTECTED CheckFunctionSupported : BOOL
VAR_IN_OUT
  /// Robot assignment of function
  AxesGroup : AxesGroup; 
END_VAR
                  CheckFunctionSupported := AxesGroup.State.RobotData.RCSupportedFunctions.SetTriggerError;

IF ( NOT CheckFunctionSupported )
THEN
  // call base implementation for set error and create log entry
  SUPER^.CheckFunctionSupported(AxesGroup := AxesGroup);
END_IF
                
END_METHOD

METHOD PROTECTED CheckParameterChanged : BOOL
VAR_IN_OUT
  /// Robot assignment of function
  AxesGroup    : AxesGroup; 
END_VAR
                  // Check ParCmd Size is > 0, because MemCmp does not work correctly with size = 0
IF (SIZEOF(ParCmd) = 0) OR (_stepCmd = 0)
THEN 
  RETURN;
END_IF

// compare memory 
_parameterChanged := ( SysDepMemCmp(pData1 := ADR(ParCmd), pData2 := ADR(_parCmd), DataLen := SIZEOF(ParCmd)) <> RobotLibraryConstants.OK );

// check parameter valid ?
_parameterValid   := CheckParameterValid( AxesGroup := AxesGroup );

IF ((  _parameterChanged        )  AND 
    (  _parameterValid          )) OR
    (  _parameterUpdateInternal )  
THEN  
  // Create log entry for parameter changed event
  CreateLogMessagePara1 ( Timestamp   := AxesGroup.State.SystemTime,
                          MessageType := MessageType.CMD,
                          Severity    := Severity.DEBUG,
                          MessageCode := 0,
                          MessageText := 'NotifyParameterChanged Event {1}',
                          Para1       :=  '' );

  // reset internal flag for send parameter update
 _parameterUpdateInternal := FALSE;
  // update internal copy of parameters 
 _parCmd := ParCmd;
  // inc parameter sequence
 _command.ParSeq := _command.ParSeq + 1;
  // update command data  
  CommandData := CreateCommandPayload(AxesGroup := AxesGroup); // ( Access via reference to rCommandFB in ACR )
  // notify active command register 
  AxesGroup.Acyclic.ActiveCommandRegister.NotifyParameterChanged := _uniqueID;
END_IF
                
END_METHOD

METHOD PROTECTED CheckParameterValid : BOOL
VAR_IN_OUT
  /// Robot assignment of function
  AxesGroup : AxesGroup; 
END_VAR
VAR
  /// internal index for loops
 _idx : DINT;
END_VAR
                  CheckParameterValid := TRUE;

// Check ParCmd.ProcessingMode defined ? 
IF (( ProcessingMode < ProcessingModeEnum.BUFFERED         ) AND
    ( ProcessingMode > ProcessingModeEnum.TRIGGER_MULTIPLE ))
THEN
  // Parameter not valid
  CheckParameterValid := FALSE;
  // Set error
  SetError( ErrorID := RobotLibraryErrorIdEnum.ERR_PROCESSINGMODE_NOT_DEFINED, Overwrite := TRUE );
  // Create log entry
  CreateLogMessagePara1 ( Timestamp   := AxesGroup.State.SystemTime,
                          MessageType := MessageType.CMD,
                          Severity    := Severity.ERROR,
                          MessageCode := ErrorID,
                          MessageText := 'Invalid Parameter ParCmd.ProcessingMode = {1}',
                          Para1       := PROCESSING_MODE_TO_STRING(ProcessingMode));
  RETURN;                          
END_IF

// Check ProcessingMode valid ? 
IF (( ProcessingMode <> ProcessingModeEnum.DEACTIVATE       ) AND 
    ( ProcessingMode <> ProcessingModeEnum.TRIGGER_ONCE     ) AND  
    ( ProcessingMode <> ProcessingModeEnum.TRIGGER_MULTIPLE ))  
THEN
  // Parameter not valid
  CheckParameterValid := FALSE;
  // Set error
  SetError( ErrorID := RobotLibraryErrorIdEnum.ERR_PROCESSINGMODE_NOT_ALLOWED, Overwrite := TRUE );
  // Create log entry
  CreateLogMessagePara1 ( Timestamp   := AxesGroup.State.SystemTime,
                          MessageType := MessageType.CMD,
                          Severity    := Severity.ERROR,
                          MessageCode := ErrorID,
                          MessageText := 'Invalid Parameter ProcessingMode = {1}',
                          Para1       := PROCESSING_MODE_TO_STRING(ProcessingMode));
  RETURN;                          
END_IF


// Check ParCmd.ErrorTriggerMode valid ? 
IF (( ParCmd.Mode <> ErrorTriggerMode.ANY_COMMAND                    ) AND
    ( ParCmd.Mode <> ErrorTriggerMode.GENERAL_COMMANDS               ) AND
    ( ParCmd.Mode <> ErrorTriggerMode.ADMINISTRATIVE_COMMANDS        ) AND
    ( ParCmd.Mode <> ErrorTriggerMode.MOVE_COMMANDS                  ) AND
    ( ParCmd.Mode <> ErrorTriggerMode.PERIPHERY_COMMANDS             ) AND
    ( ParCmd.Mode <> ErrorTriggerMode.EXTENDED_COMMANDS              ) AND
    ( ParCmd.Mode <> ErrorTriggerMode.SPECIFIC_COMMAND_OR_RI_MESSAGE ) AND
    ( ParCmd.Mode <> ErrorTriggerMode.SPECIFIC_RC_OR_RA_MESSAGE_CODE ) AND
    ( ParCmd.Mode <> ErrorTriggerMode.ANY_RI_MESSAGE_CODE            ) AND
    ( ParCmd.Mode <> ErrorTriggerMode.ANY_RC_OR_RA_MESSAGE_CODE      ))
    
THEN
  // Parameter not valid
  CheckParameterValid := FALSE;
  // Set error
  SetError( ErrorID := RobotLibraryErrorIdEnum.ERR_INVALID_PAR_CMD, Overwrite := TRUE );
  // Create log entry
  CreateLogMessagePara1 ( Timestamp   := AxesGroup.State.SystemTime,
                          MessageType := MessageType.CMD,
                          Severity    := Severity.ERROR,
                          MessageCode := ErrorID,
                          MessageText := 'Invalid Parameter ParCmd.ErrorTriggerMode = {1}',
                          Para1       := ERROR_TRIGGER_MODE_TO_STRING(ParCmd.Mode));
  RETURN;                          
END_IF

FOR _idx := 0 TO RobotLibraryParameter.MESSAGE_CODES_MAX
DO
  // Check ParCmd.MessageCodes[x] valid ? 
  IF  (( ParCmd.MessageCodes[_idx] <             0 ) OR
       ( ParCmd.MessageCodes[_idx] >  16#FFFF_FFFF ))     
  THEN
    // Parameter not valid
    CheckParameterValid := FALSE;
    // Set error
    SetError( ErrorID := RobotLibraryErrorIdEnum.ERR_INVALID_PAR_CMD, Overwrite := TRUE );
    // Create log entry
    CreateLogMessagePara2 ( Timestamp   := AxesGroup.State.SystemTime,
                            MessageType := MessageType.CMD,
                            Severity    := Severity.ERROR,
                            MessageCode := ErrorID,
                            MessageText := 'Invalid Parameter ParCmd.MessageCodes[{2}] = {1}',
                            Para1       := DWORD_TO_STRING(ParCmd.MessageCodes[_idx]),
                            Para2       := DINT_TO_STRING(_idx));
    EXIT;
    RETURN;
  END_IF
END_FOR


// Check ParCmd.IncludeParameterValidation
// -> no plausibility check for boolean


// Check ParCmd.ListenerID valid ? 
IF  (( ParCmd.ListenerID <    0 ) OR
     ( ParCmd.ListenerID >  127 ))     
THEN
  // Parameter not valid
  CheckParameterValid := FALSE;
  // Set error
  SetError( ErrorID := RobotLibraryErrorIdEnum.ERR_INVALID_PAR_CMD, Overwrite := TRUE );
  // Create log entry
  CreateLogMessagePara1 ( Timestamp   := AxesGroup.State.SystemTime,
                          MessageType := MessageType.CMD,
                          Severity    := Severity.ERROR,
                          MessageCode := ErrorID,
                          MessageText := 'Invalid Parameter ParCmd.ListenerID = {1}',
                          Para1       := SINT_TO_STRING(ParCmd.ListenerID));
  RETURN;
END_IF

// Check ParCmd.EmitterID valid ? 
IF  (( ParCmd.EmitterID < -127 ) OR
     ( ParCmd.EmitterID >  127 ))     
THEN
  // Parameter not valid
  CheckParameterValid := FALSE;
  // Set error
  SetError( ErrorID := RobotLibraryErrorIdEnum.ERR_INVALID_PAR_CMD, Overwrite := TRUE );
  // Create log entry
  CreateLogMessagePara1 ( Timestamp   := AxesGroup.State.SystemTime,
                          MessageType := MessageType.CMD,
                          Severity    := Severity.ERROR,
                          MessageCode := ErrorID,
                          MessageText := 'Invalid Parameter ParCmd.EmitterID = {1}',
                          Para1       := SINT_TO_STRING(ParCmd.EmitterID));
  RETURN;
END_IF

                
END_METHOD

METHOD INTERNAL CreateCommandPayload : RobotLibraryCommandDataFB
VAR_IN_OUT
  /// Robot assignment of function
  AxesGroup : AxesGroup; 
END_VAR
VAR
  /// internal index for loops
 _idx          : DINT;
  /// Parameter count
 _parameterCnt : DINT;
END_VAR
// Table 6-598: Sent CMD payload (PLC to RC) of "SetTriggerError"
// --------------------------
// Header
// --------------------------
// Byte 00 : UINT  - Type HB     
// Byte 01 :       - Type LB    
// Byte 02 : USINT - Reserve | ExecutionMode
// Byte 03 : USINT - ParSeq  | Priority
// --------------------------
// Datablock
// --------------------------
// Byte 00 : UINT  Type;
// Byte 01 :       Type;
// Byte 02 : USINT Reserved ExecutionMode;
// Byte 03 : USINT ParSeq Priority;
// Byte 04 : SINT  EmitterID[0];
// Byte 05 : SINT  EmitterID[1];
// Byte 06 : SINT  EmitterID[2];
// Byte 07 : SINT  EmitterID[3];
// Byte 08 : SINT  ListenerID;
// Byte 09 : BYTE  Reserved;
// Byte 10 : SINT  Mode;
// Byte 11 : BOOL  IncludeParameterValidation;
// Byte 12 : DWORD MessageCode[0];
// Byte 13 :       MessageCode[0];
// Byte 14 :       MessageCode[0];
// Byte 15 :       MessageCode[0];
// Byte 16 : DWORD MessageCode[1];
// Byte 17 :       MessageCode[1];
// Byte 18 :       MessageCode[1];
// Byte 19 :       MessageCode[1];
// Byte 20 : DWORD MessageCode[2];
// Byte 21 :       MessageCode[2];
// Byte 22 :       MessageCode[2];
// Byte 23 :       MessageCode[2];
// Byte 24 : DWORD MessageCode[3];
// Byte 25 :       MessageCode[3];
// Byte 26 :       MessageCode[3];
// Byte 27 :       MessageCode[3];
// Byte 28 : DWORD MessageCode[4];
// Byte 29 :       MessageCode[4];
// Byte 30 :       MessageCode[4];
// Byte 31 :       MessageCode[4];
// Byte 32 : DWORD MessageCode[5];
// Byte 33 :       MessageCode[5];
// Byte 34 :       MessageCode[5];
// Byte 35 :       MessageCode[5];
// Byte 36 : DWORD MessageCode[6];
// Byte 37 :       MessageCode[6];
// Byte 38 :       MessageCode[6];
// Byte 39 :       MessageCode[6];
// Byte 40 : DWORD MessageCode[7];
// Byte 41 :       MessageCode[7];
// Byte 42 :       MessageCode[7];
// Byte 43 :       MessageCode[7];
// Byte 44 : DWORD MessageCode[8];
// Byte 45 :       MessageCode[8];
// Byte 46 :       MessageCode[8];
// Byte 47 :       MessageCode[8];
// Byte 48 : DWORD MessageCode[9];
// Byte 49 :       MessageCode[9];
// Byte 50 :       MessageCode[9];
// Byte 51 :       MessageCode[9];
// Byte 52 : DWORD MessageCode[10];
// Byte 53 :       MessageCode[10];
// Byte 54 :       MessageCode[10];
// Byte 55 :       MessageCode[10];
// Byte 56 : DWORD MessageCode[11];
// Byte 57 :       MessageCode[11];
// Byte 58 :       MessageCode[11];
// Byte 59 :       MessageCode[11];
// Byte 60 : DWORD MessageCode[12];
// Byte 61 :       MessageCode[12];
// Byte 62 :       MessageCode[12];
// Byte 63 :       MessageCode[12];
// Byte 64 : DWORD MessageCode[13];
// Byte 65 :       MessageCode[13];
// Byte 66 :       MessageCode[13];
// Byte 67 :       MessageCode[13];
// Byte 68 : DWORD MessageCode[14];
// Byte 69 :       MessageCode[14];
// Byte 70 :       MessageCode[14];
// Byte 71 :       MessageCode[14];
// Byte 72 : DWORD MessageCode[15];
// Byte 73 :       MessageCode[15];
// Byte 74 :       MessageCode[15];
// Byte 75 :       MessageCode[15];
                  // set command parameter 
_command.CmdTyp                    :=  CmdType.SetTriggerError;
_command.ExecMode                  :=  ExecMode;
_command.ParSeq                    := _command.ParSeq;
_command.Priority                  :=  Priority;

_command.EmitterID[0]              := _parCmd.EmitterID;
_command.EmitterID[1]              := 0;
_command.EmitterID[2]              := 0;
_command.EmitterID[3]              := 0;
_command.ListenerID                := _parCmd.ListenerID;
_command.Reserve                   := 0;
_command.Mode                      := _parCmd.Mode;
_command.IncludeParameterValidation:= _parCmd.IncludeParameterValidation;
_command.MessageCodes              := _parCmd.MessageCodes;


// copy command data to header
_cmdHeader := _command;
// call base implementation to copy header to payload buffer
CreateCommandPayload := SUPER^.CreateCommandPayload(AxesGroup := AxesGroup);


FOR _idx := 0 TO 3 
DO
  // Check parameter must be added ? 
  IF ( CheckAddParameter(CreateCommandPayload.PayloadPtr))
  THEN
    // add command.EmitterID[x]
    CreateCommandPayload.AddSint(_command.EmitterID[_idx]);
    // inc parameter counter
   _parameterCnt := _parameterCnt + 1;  
  END_IF
END_FOR


// Check parameter must be added ? 
IF ( CheckAddParameter(CreateCommandPayload.PayloadPtr))
THEN
  // add command.ListenerID
  CreateCommandPayload.AddSint(_command.ListenerID);
  // inc parameter counter
 _parameterCnt := _parameterCnt + 1;  
END_IF


// Check parameter must be added ? 
IF ( CheckAddParameter(CreateCommandPayload.PayloadPtr))
THEN
  // add command.Reserve
  CreateCommandPayload.AddSint(_command.Reserve);
  // inc parameter counter
 _parameterCnt := _parameterCnt + 1;  
END_IF


// Check parameter must be added ? 
IF ( CheckAddParameter(CreateCommandPayload.PayloadPtr))
THEN
  // add command.Mode
  CreateCommandPayload.AddSint(_command.Mode);
  // inc parameter counter
 _parameterCnt := _parameterCnt + 1;  
END_IF


// Check parameter must be added ? 
IF ( CheckAddParameter(CreateCommandPayload.PayloadPtr))
THEN
  // add command.IncludeParameterValidation
  CreateCommandPayload.AddBool(_command.IncludeParameterValidation);
  // inc parameter counter
 _parameterCnt := _parameterCnt + 1;  
END_IF


FOR _idx := 0 TO RobotLibraryParameter.MESSAGE_CODES_MAX
DO
  // Check parameter must be added ? 
  IF ( CheckAddParameter(CreateCommandPayload.PayloadPtr))
  THEN
    // add command.MessageCodes[_idx]
    CreateCommandPayload.AddDword(_command.MessageCodes[_idx]);
    // inc parameter counter
   _parameterCnt := _parameterCnt + 1;  
  END_IF
END_FOR


// Create logging
CreateCommandPayloadLog(AxesGroup := AxesGroup, ParameterCnt := _parameterCnt);
                
END_METHOD

METHOD INTERNAL CreateCommandPayloadLog
VAR_IN_OUT
  /// Robot assignment of function
  AxesGroup : AxesGroup; 
END_VAR
VAR_INPUT
  /// Parameter count
  ParameterCnt : DINT;
END_VAR
VAR 
  /// internal index for loops
 _idx : DINT;
END_VAR
                  // Create log entry for Parameter start
CreateLogMessagePara1 ( Timestamp   := AxesGroup.State.SystemTime,
                        MessageType := MessageType.CMD,
                        Severity    := Severity.DEBUG,
                        MessageCode := 0,
                        MessageText := 'Create command payload with {1} parameter(s) :',
                        Para1       := DINT_TO_STRING(ParameterCnt));
  
// Create log entry for EmitterID[x]
FOR _idx := 0 TO 3
DO
  // Return if no parameter is remaining...
  IF ( ParameterCnt = 0 ) THEN RETURN; END_IF
  // dec remaining parameter(s)                        
  ParameterCnt := ParameterCnt - 1;
  // Create log entry for Command.EmitterID
  CreateLogMessagePara2 ( Timestamp   := AxesGroup.State.SystemTime,
                          MessageType := MessageType.CMD,
                          Severity    := Severity.DEBUG,
                          MessageCode := 0,
                          MessageText := 'Command.EmitterID[{2}] = {1}',
                          Para1       :=  SINT_TO_STRING(_command.EmitterID[_idx]),
                          Para2       :=  DINT_TO_STRING(_idx));
END_FOR


// Return if no parameter is remaining...
IF ( ParameterCnt = 0 ) THEN RETURN; END_IF
// dec remaining parameter(s)                        
ParameterCnt := ParameterCnt - 1;
// Create log entry for ListenerID
CreateLogMessagePara1 ( Timestamp   := AxesGroup.State.SystemTime,
                        MessageType := MessageType.CMD,
                        Severity    := Severity.DEBUG,
                        MessageCode := 0,
                        MessageText := 'Command.ListenerID = {1}',
                        Para1       :=  SINT_TO_STRING(_command.ListenerID));
                        

// Return if no parameter is remaining...
IF ( ParameterCnt = 0 ) THEN RETURN; END_IF
// dec remaining parameter(s)                        
ParameterCnt := ParameterCnt - 1;
// Create log entry for Reserve
CreateLogMessagePara1 ( Timestamp   := AxesGroup.State.SystemTime,
                        MessageType := MessageType.CMD,
                        Severity    := Severity.DEBUG,
                        MessageCode := 0,
                        MessageText := 'Command.Reserve = {1}',
                        Para1       :=  SINT_TO_STRING(_command.Reserve));


// Return if no parameter is remaining...
IF ( ParameterCnt = 0 ) THEN RETURN; END_IF
// dec remaining parameter(s)                        
ParameterCnt := ParameterCnt - 1;
// Create log entry for Mode
CreateLogMessagePara1 ( Timestamp   := AxesGroup.State.SystemTime,
                        MessageType := MessageType.CMD,
                        Severity    := Severity.DEBUG,
                        MessageCode := 0,
                        MessageText := 'Command.Mode = {1}',
                        Para1       :=  ERROR_TRIGGER_MODE_TO_STRING(_command.Mode));


// Return if no parameter is remaining...
IF ( ParameterCnt = 0 ) THEN RETURN; END_IF
// dec remaining parameter(s)                        
ParameterCnt := ParameterCnt - 1;
// Create log entry for IncludeParameterValidation
CreateLogMessagePara1 ( Timestamp   := AxesGroup.State.SystemTime,
                        MessageType := MessageType.CMD,
                        Severity    := Severity.DEBUG,
                        MessageCode := 0,
                        MessageText := 'Command.IncludeParameterValidation = {1}',
                        Para1       :=  BOOL_TO_STRING(_command.IncludeParameterValidation));

// add command.MessageCodes[_idx]
FOR _idx := 0 TO RobotLibraryParameter.MESSAGE_CODES_MAX
DO
  // Return if no parameter is remaining...
  IF ( ParameterCnt = 0 ) THEN RETURN; END_IF
  // dec remaining parameter(s)                        
  ParameterCnt := ParameterCnt - 1;
  // Create log entry for Command.MessageCodes
  CreateLogMessagePara2 ( Timestamp   := AxesGroup.State.SystemTime,
                          MessageType := MessageType.CMD,
                          Severity    := Severity.DEBUG,
                          MessageCode := 0,
                          MessageText := 'Command.MessageCodes[{2}] = {1}',
                          Para1       :=  DWORD_TO_STRING(_command.MessageCodes[_idx]),
                          Para2       :=  DINT_TO_STRING(_idx));
  
END_FOR
                
END_METHOD

METHOD FB_init : BOOL
VAR_INPUT
  /// if TRUE, the retain variables are initialized (warm start / cold start)
  bInitRetains : BOOL; 
  /// if TRUE, the instance afterwards gets moved into the copy code (online change)
  bInCopyCode  : BOOL;  
END_VAR
                  MyType := 'MC_SetTriggerErrorFB';

ExecMode       := ExecutionMode.PARALLEL;
Priority       := PriorityLevel.NORMAL;
ProcessingMode := ProcessingModeEnum.TRIGGER_ONCE;
                
END_METHOD

METHOD PROTECTED OnApplyOutCmd
VAR_INPUT
  /// Command message state
  State : CmdMessageState;
END_VAR
                  IF ( State = CmdMessageState.EMPTY ) 
THEN
  // Reset command outputs
  SysDepMemSet(pDest := ADR(OutCmd), Value := 0, DataLen := SIZEOF(OutCmd));         
END_IF

IF (( State = CmdMessageState.ACTIVE ) OR
    ( State = CmdMessageState.DONE   ))
THEN
  // Update results
  OutCmd.FollowID          := _response.OriginID;
  OutCmd.OriginID          := _response.OriginID;
  OutCmd.InvocationCounter := _response.InvocationCounter;
END_IF
                
END_METHOD

METHOD PROTECTED OnExecRun : DINT
VAR_IN_OUT
  /// Robot assignment of function
  AxesGroup : AxesGroup; 
END_VAR
                  // call base implementation
SUPER^.OnExecRun(AxesGroup := AxesGroup);

CASE _stepCmd OF
  
  00:  IF ( _execute_R.Q ) AND ( NOT Error)  
       THEN
         // Check function is supported and parameter are valid ?
         IF (( CheckFunctionSupported( AxesGroup := AxesGroup )) AND
             ( CheckParameterValid   ( AxesGroup := AxesGroup )))
         THEN      
           // set busy flag
           Busy := TRUE;
           // Reset command outputs
           SysDepMemSet(pDest := ADR(OutCmd), Value := 0, DataLen := SIZEOF(OutCmd));         
           // apply command parameter
          _parCmd := ParCmd;
           // init parameter sequence
          _command.ParSeq := 1;
           // create command data
           CommandData := CreateCommandPayload(AxesGroup := AxesGroup);
           // Add command to active command register
          _uniqueID := AxesGroup.Acyclic.ActiveCommandRegister.AddCmd( pCommandFB := ADR(THIS^ ));     
           // set timeout
           SetTimeout(PT := _timeoutCmd, rTimer := _timerCmd);
           // inc step counter
          _stepCmd := _stepCmd + 1;
         END_IF 
       END_IF
     

  01:  // Wait for responce received
       IF ( _responseReceived )
       THEN
         // reset response received flag
        _responseReceived := FALSE;
         // update state flags
         OnUpdateStateFlags(_response.State);
         // update state flags
         OnApplyOutCmd(_response.State);
                
         // Done, Aborted or Error ?
         IF (_response.State >= CmdMessageState.DONE )
         THEN
           // set timeout
           SetTimeout(PT := _timeoutCmd, rTimer := _timerCmd);
           // inc step counter
          _stepCmd := _stepCmd + 1; 
         END_IF
       END_IF


  02: IF ( NOT Execute)
      THEN
        Reset();
      END_IF     

ELSE
  // invalid step
  SetError( ErrorID := RobotLibraryErrorIdEnum.ERR_INVALID_STEP, Overwrite := TRUE );
END_CASE


// Reset FB
IF ( NOT Execute )
THEN
  Reset();
END_IF
                
END_METHOD

METHOD PROTECTED OnUpdateStateFlags
VAR_INPUT
  /// Command message state
  State : CmdMessageState;
END_VAR
                  // Reset State flags
Done               := FALSE;
MonitoringActive   := FALSE;

CASE State OF

  // No operation or process is active
  CmdMessageState.EMPTY               :;
  // Created but not yet started
  CmdMessageState.CREATED             :;
  // Buffered and awaiting execution
  CmdMessageState.BUFFERED            : CommandBuffered    := TRUE;                                        
  // Buffered in planner for future execution
  CmdMessageState.BUFFERED_IN_PLANNER : CommandBuffered    := TRUE; 
  // Currently active and in progress
  CmdMessageState.ACTIVE              : MonitoringActive   := TRUE;                                  
  // Interrupted and awaiting continuation
  CmdMessageState.INTERRUPTED         :;     
  // Requested for abort
  CmdMessageState.ABORT_REQUEST       :;
  // Successfully completed
  CmdMessageState.DONE                : Done               := TRUE;
                                        Busy               := FALSE;
  // Aborted before completion
  CmdMessageState.ABORTED             : Busy               := FALSE;
  // Encountered an error during execution
  CmdMessageState.ERROR               : Error              := TRUE;
                                        Busy               := FALSE;
END_CASE
                
END_METHOD

METHOD INTERNAL ParseResponsePayload : DINT
VAR_INPUT
  /// Response data
  ResponseData : RobotLibraryResponseDataFB;
  /// Timestamp
  Timestamp    : SystemTime;  
END_VAR
VAR
  /// Parameter count
 _parameterCnt : DINT;
END_VAR
// 6-599: Received CMD payload (RC to PLC) of "SetTriggerError" 
// --------------------------
// Header
// --------------------------
// Byte 00 : USINT   - ParSeq | State     
// Byte 01 : SINT    - AlarmMessageSeverity    
// Byte 02 : UINT    - AlarmMessageCode HB
// Byte 03 :         - AlarmMessageCode LB
// --------------------------
// Datablock
// --------------------------
// Byte 04 : USINT   - InvocationCounter
// Byte 05 : SINT    - Reserve
// Byte 06 : INT     - OriginID LW HB
// Byte 07 :         - OriginID LW LB
                  // call base implementation to parse the header from payload buffer
ResponseData.PayloadPtr := SUPER^.ParseResponsePayload(ResponseData := ResponseData, Timestamp := Timestamp);

// copy parsed header to response
_response.ParSeq               := _rspHeader.ParSeq;
_response.State                := _rspHeader.State;
_response.AlarmMessageSeverity := _rspHeader.AlarmMessageSeverity;
_response.AlarmMessageCode     := _rspHeader.AlarmMessageCode;


// Check payload remaining ? 
IF ( ResponseData.IsPayloadRemaining)
THEN  
  // Get Response.InvocationCounter
 _response.InvocationCounter := ResponseData.GetUsint();
  // inc parameter counter
 _parameterCnt := _parameterCnt + 1;
END_IF


// Check payload remaining ? 
IF ( ResponseData.IsPayloadRemaining)
THEN  
  // Get Response.Reserve
 _response.Reserve := ResponseData.GetSint();
  // inc parameter counter
 _parameterCnt := _parameterCnt + 1;
END_IF


// Check payload remaining ? 
IF ( ResponseData.IsPayloadRemaining)
THEN  
  // Get Response.OriginID
 _response.OriginID := ResponseData.GetInt();
  // inc parameter counter
 _parameterCnt := _parameterCnt + 1;
END_IF


// Create logging
ParseResponsePayloadLog(ResponseData := ResponseData, Timestamp := Timestamp, ParameterCnt := _parameterCnt);
                
END_METHOD

METHOD INTERNAL ParseResponsePayloadLog
VAR_INPUT
  /// Response data
  ResponseData : RobotLibraryResponseDataFB;
  /// Timestamp
  Timestamp    : SystemTime;  
  /// Parameter count
  ParameterCnt : DINT;
END_VAR
                  // Create log entry for Parameter start
CreateLogMessagePara1 ( Timestamp   := Timestamp,
                        MessageType := MessageType.CMD,
                        Severity    := Severity.DEBUG,
                        MessageCode := 0,
                        MessageText := '{1} parameter(s) to parse from the response data:',
                        Para1       := DINT_TO_STRING(ParameterCnt));
                        

// Return if no parameter is remaining...
IF ( ParameterCnt = 0 ) THEN RETURN; END_IF
// dec remaining parameter(s)                        
ParameterCnt := ParameterCnt - 1;
// Create log entry for InvocationCounter
CreateLogMessagePara1 ( Timestamp   := Timestamp,
                        MessageType := MessageType.CMD,
                        Severity    := Severity.DEBUG,
                        MessageCode := 0,
                        MessageText := 'Response.InvocationCounter = {1}',
                        Para1       :=  USINT_TO_STRING(_response.InvocationCounter));


// Return if no parameter is remaining...
IF ( ParameterCnt = 0 ) THEN RETURN; END_IF
// dec remaining parameter(s)                        
ParameterCnt := ParameterCnt - 1;
// Create log entry for Reserve
CreateLogMessagePara1 ( Timestamp   := Timestamp,
                        MessageType := MessageType.CMD,
                        Severity    := Severity.DEBUG,
                        MessageCode := 0,
                        MessageText := 'Response.Reserve = {1}',
                        Para1       :=  SINT_TO_STRING(_response.Reserve));


// Return if no parameter is remaining...
IF ( ParameterCnt = 0 ) THEN RETURN; END_IF
// dec remaining parameter(s)                        
ParameterCnt := ParameterCnt - 1;
// Create log entry for OriginID
CreateLogMessagePara1 ( Timestamp   := Timestamp,
                        MessageType := MessageType.CMD,
                        Severity    := Severity.DEBUG,
                        MessageCode := 0,
                        MessageText := 'Response.OriginID = {1}',
                        Para1       :=  INT_TO_STRING(_response.OriginID));
                
END_METHOD

METHOD PROTECTED Reset : DINT
VAR_INPUT
END_VAR
                  Reset := SUPER^.Reset();

Done             := FALSE;
Busy             := FALSE;
CommandBuffered  := FALSE;
MonitoringActive := FALSE;
                
END_METHOD
END_FUNCTION_BLOCK

/// Trigger "Actions" based on physical events (e.g. force limit reached)
FUNCTION_BLOCK MC_SetTriggerLimitFB EXTENDS RobotLibraryBaseExecuteFB
// ------------------------------------------------------------------------- 
//  SRCI Robot Library                                                
// ------------------------------------------------------------------------- 
//                                                                           
//  Object:      SetTriggerLimitFB                                       
//  Author:      Thorsten Brach                                                
//  Date:        2024-06-01
//
//  Description:                                              
//   
//                                                                           
//  Copyright: 
//    (C) 2024 Thorsten Brach. All rights reserved                                                                                                                                            
//             Licensed under the MIT License.
//                                                                           
//  Disclaimer:                                                                           
//    This project is provided without any guarantee and can be used for   
//    private and commercial purposes. Any use is at the user’s 
//    own risk and responsibility.
//
// -------------------------------------------------------------------------
VAR_INPUT
  /// command parameter 
  ParCmd           : SetTriggerLimitParCmd;
  /// Processing mode
  ProcessingMode   : ProcessingMode;
END_VAR
VAR_OUTPUT
  /// TRUE, while the following outputs return valid values:
  /// • Data
  Valid            : BOOL;
  /// Command is transferred and confirmed by the RC
  CommandBuffered  : BOOL;
  /// TRUE, when the monitoring of the input parameter values is active.
  MonitoringActive : BOOL;
  /// command results
  OutCmd           : SetTriggerLimitOutCmd;     
END_VAR

VAR
  /// internal copy of command parameter 
 _parCmd           : SetTriggerLimitParCmd;
  /// command data to send
 _command          : SetTriggerLimitSendData;
  /// response data received
 _response         : SetTriggerLimitRecvData;      
END_VAR

            SUPER^(AxesGroup := AxesGroup);
          

METHOD INTERNAL CheckAddParameter : BOOL
VAR_INPUT
  /// Payload pointer
  PayloadPtr : UDINT;
END_VAR
VAR
  /// Payload as byte array
  Payload    : ARRAY [1..SIZEOF(_command)] OF BYTE;
  /// Null Byte array 
  Null       : ARRAY [1..SIZEOF(_command)] OF BYTE;
  /// Data length to compare
  DataLen    : UDINT;
END_VAR
                  // Payload pointer must be decreased by one byte, because ADR(Payload) is already one byte !
PayloadPtr := LIMIT (0, PayloadPtr - 1, SIZEOF(Payload) -1);
// Convert command struct to payload array
SysDepMemCpy( pDest := ADR(Payload), pSrc := ADR(_command), DataLen := SIZEOF(_command));
// Calculate the data length to compare - at least one byte must be compared !
DataLen := LIMIT(1, SIZEOF(Payload) - PayloadPtr, SIZEOF(Payload)); 
// Compare Payload-Array with Null-Byte-Array
CheckAddParameter := SysDepMemCmp( pData1 := ADR(Payload) + PayloadPtr , pData2 := ADR(Null), DataLen := DataLen) <>  RobotLibraryConstants.OK ;
                
END_METHOD

METHOD PROTECTED CheckFunctionSupported : BOOL
VAR_IN_OUT
  /// Robot assignment of function
  AxesGroup : AxesGroup; 
END_VAR
                  CheckFunctionSupported := AxesGroup.State.RobotData.RCSupportedFunctions.SetTriggerLimit;

IF ( NOT CheckFunctionSupported )
THEN
  // call base implementation for set error and create log entry
  SUPER^.CheckFunctionSupported(AxesGroup := AxesGroup);
END_IF
                
END_METHOD

METHOD PROTECTED CheckParameterChanged : BOOL
VAR_IN_OUT
  /// Robot assignment of function
  AxesGroup    : AxesGroup; 
END_VAR
                  // Check ParCmd Size is > 0, because MemCmp does not work correctly with size = 0
IF (SIZEOF(ParCmd) = 0) OR (_stepCmd = 0)
THEN 
  RETURN;
END_IF

// compare memory 
_parameterChanged := ( SysDepMemCmp(pData1 := ADR(ParCmd), pData2 := ADR(_parCmd), DataLen := SIZEOF(ParCmd)) <> RobotLibraryConstants.OK );

// check parameter valid ?
_parameterValid   := CheckParameterValid( AxesGroup := AxesGroup );

IF ((  _parameterChanged        )  AND 
    (  _parameterValid          )) OR
    (  _parameterUpdateInternal )  
THEN  
  // Create log entry for parameter changed event
  CreateLogMessagePara1 ( Timestamp   := AxesGroup.State.SystemTime,
                          MessageType := MessageType.CMD,
                          Severity    := Severity.DEBUG,
                          MessageCode := 0,
                          MessageText := 'NotifyParameterChanged Event {1}',
                          Para1       :=  '' );

  // reset internal flag for send parameter update
 _parameterUpdateInternal := FALSE;
  // update internal copy of parameters 
 _parCmd := ParCmd;
  // inc parameter sequence
 _command.ParSeq := _command.ParSeq + 1;
  // update command data  
  CommandData := CreateCommandPayload(AxesGroup := AxesGroup); // ( Access via reference to rCommandFB in ACR )
  // notify active command register 
  AxesGroup.Acyclic.ActiveCommandRegister.NotifyParameterChanged := _uniqueID;
  // Reset Valid output of the FB 
  Valid := FALSE;
END_IF
                
END_METHOD

METHOD PROTECTED CheckParameterValid : BOOL
VAR_IN_OUT
  /// Robot assignment of function
  AxesGroup : AxesGroup; 
END_VAR
VAR
  /// internal index for loops
 _idx : DINT;
END_VAR
                  CheckParameterValid := TRUE;

// Check ParCmd.ProcessingMode defined ? 
IF (( ProcessingMode < ProcessingModeEnum.BUFFERED         ) AND
    ( ProcessingMode > ProcessingModeEnum.TRIGGER_MULTIPLE ))
THEN
  // Parameter not valid
  CheckParameterValid := FALSE;
  // Set error
  SetError( ErrorID := RobotLibraryErrorIdEnum.ERR_PROCESSINGMODE_NOT_DEFINED, Overwrite := TRUE );
  // Create log entry
  CreateLogMessagePara1 ( Timestamp   := AxesGroup.State.SystemTime,
                          MessageType := MessageType.CMD,
                          Severity    := Severity.ERROR,
                          MessageCode := ErrorID,
                          MessageText := 'Invalid Parameter ParCmd.ProcessingMode = {1}',
                          Para1       := PROCESSING_MODE_TO_STRING(ProcessingMode));
  RETURN;                          
END_IF

